LIN {X 0,Y 200.073,Z 515.512,A -85,B 0,C 180,E1 -21845.07,E2 -21845.07} C_VEL
LIN {X 0,Y 196.542,Z 522.437,A -85,B 0,C 180,E1 -21849.049,E2 -21849.049} C_VEL
LIN {X 0,Y 193.866,Z 527.871,A -85,B 0,C 180,E1 -21853.142,E2 -21853.142} C_VEL
LIN {X 0,Y 192.041,Z 531.966,A -85,B 0,C 180,E1 -21857.316,E2 -21857.316} C_VEL
LIN {X 0,Y 190.931,Z 534.837,A -85,B 0,C 180,E1 -21861.533,E2 -21861.533} C_VEL
LIN {X 0,Y 190.385,Z 536.558,A -85,B 0,C 180,E1 -21865.766,E2 -21865.766} C_VEL
LIN {X 0,Y 190.301,Z 537.156,A -85,B 0,C 180,E1 -21870,E2 -21870} C_VEL
LIN {X 0,Y 190.444,Z 536.444,A -85,B 0,C 180,E1 -21874.869,E2 -21874.869} C_VEL
LIN {X 0,Y 190.924,Z 534.92,A -85,B 0,C 180,E1 -21878.467,E2 -21878.467} C_VEL
LIN {X 0,Y 192.016,Z 532.092,A -85,B 0,C 180,E1 -21882.686,E2 -21882.686} C_VEL
LIN {X 0,Y 193.842,Z 528.039,A -85,B 0,C 180,E1 -21886.861,E2 -21886.861} C_VEL
LIN {X 0,Y 196.544,Z 522.658,A -85,B 0,C 180,E1 -21890.951,E2 -21890.951} C_VEL
LIN {X 0,Y 199.996,Z 515.797,A -85,B 0,C 180,E1 -21894.941,E2 -21894.941} C_VEL
LIN {X 0,Y 204.38,Z 507.224,A -85,B 0,C 180,E1 -21898.777,E2 -21898.777} C_VEL
LIN {X 0,Y 208.207,Z 499.512,A -85,B 0,C 180,E1 -21901.546,E2 -21901.546} C_VEL
LIN {X 0,Y 212.272,Z 490.435,A -85,B 0,C 180,E1 -21904.252,E2 -21904.252} C_VEL
LIN {X 0,Y 216.99,Z 479.715,A -85,B 0,C 180,E1 -21906.811,E2 -21906.811} C_VEL
LIN {X 0,Y 221.502,Z 468.012,A -85,B 0,C 180,E1 -21909.094,E2 -21909.094} C_VEL
LIN {X 0,Y 226.056,Z 455.219,A -85,B 0,C 180,E1 -21911.053,E2 -21911.053} C_VEL
LIN {X 0,Y 229.873,Z 442.172,A -85,B 0,C 180,E1 -21912.681,E2 -21912.681} C_VEL
LIN {X 0,Y 233.233,Z 428.457,A -85,B 0,C 180,E1 -21914.021,E2 -21914.021} C_VEL
LIN {X 0,Y 236.191,Z 413.431,A -85,B 0,C 180,E1 -21915.116,E2 -21915.116} C_VEL
LIN {X 0,Y 238.192,Z 399.868,A -85,B 0,C 180,E1 -21915.835,E2 -21915.835} C_VEL
LIN {X 0,Y 239.696,Z 384.094,A -85,B 0,C 180,E1 -21916.372,E2 -21916.372} C_VEL
LIN {X 0,Y 244.254,Z 312.757,A -85,B 0,C 180,E1 -21918.264,E2 -21918.264} C_VEL
LIN {X 0,Y 244.009,Z 311.507,A -85,B 0,C 180,E1 -21918.383,E2 -21918.383} C_VEL
LIN {X 0,Y 240.206,Z 303.509,A -85,B 0,C 180,E1 -21919.784,E2 -21919.784} C_VEL
LIN {X 0,Y 232.844,Z 290.889,A -85,B 0,C 180,E1 -21922.617,E2 -21922.617} C_VEL
LIN {X 0,Y 226.849,Z 281.57,A -85,B 0,C 180,E1 -21925.165,E2 -21925.165} C_VEL
LIN {X 0,Y 221.021,Z 273.151,A -85,B 0,C 180,E1 -21927.918,E2 -21927.918} C_VEL
LIN {X 0,Y 217.818,Z 268.869,A -85,B 0,C 180,E1 -21929.572,E2 -21929.572} C_VEL
LIN {X 0,Y 214.771,Z 264.799,A -85,B 0,C 180,E1 -21931.274,E2 -21931.274} C_VEL
LIN {X 0,Y 211.832,Z 260.873,A -85,B 0,C 180,E1 -21933.059,E2 -21933.059} C_VEL
LIN {X 0,Y 208.609,Z 257.265,A -85,B 0,C 180,E1 -21935.161,E2 -21935.161} C_VEL
LIN {X 0,Y 207.468,Z 255.378,A -85,B 0,C 180,E1 -21936.015,E2 -21936.015} C_VEL
LIN {X 0,Y 204.837,Z 253.006,A -85,B 0,C 180,E1 -21937.959,E2 -21937.959} C_VEL
LIN {X 0,Y 203.12,Z 250.05,A -85,B 0,C 180,E1 -21939.492,E2 -21939.492} C_VEL
LIN {X 0,Y 200.172,Z 247.881,A -85,B 0,C 180,E1 -21942.158,E2 -21942.158} C_VEL
LIN {X 0,Y 198.485,Z 244.934,A -85,B 0,C 180,E1 -21944.139,E2 -21944.139} C_VEL
LIN {X 0,Y 198.171,Z 244.119,A -85,B 0,C 180,E1 -21944.574,E2 -21944.574} C_VEL
LIN {X 0,Y 195.148,Z 242.441,A -85,B 0,C 180,E1 -21948.575,E2 -21948.575} C_VEL
LIN {X 0,Y 193.097,Z 238.68,A -85,B 0,C 180,E1 -21953.338,E2 -21953.338} C_VEL
LIN {X 0,Y 192.983,Z 238.059,A -85,B 0,C 180,E1 -21953.99,E2 -21953.99} C_VEL
LIN {X 0,Y 193.259,Z 238.03,A -85,B 0,C 180,E1 -21957.916,E2 -21957.916} C_VEL
LIN {X 0,Y 193.439,Z 238,A -85,B 0,C 180,E1 -21960,E2 -21960} C_VEL
LIN {X 0,Y 192.97,Z 238.063,A -85,B 0,C 180,E1 -21965.224,E2 -21965.224} C_VEL
LIN {X 0,Y 193.024,Z 238.361,A -85,B 0,C 180,E1 -21966.008,E2 -21966.008} C_VEL
LIN {X 0,Y 193.993,Z 240.918,A -85,B 0,C 180,E1 -21968.857,E2 -21968.857} C_VEL
LIN {X 0,Y 196.391,Z 243.419,A -85,B 0,C 180,E1 -21972.924,E2 -21972.924} C_VEL
LIN {X 0,Y 198.288,Z 244.285,A -85,B 0,C 180,E1 -21975.218,E2 -21975.218} C_VEL
LIN {X 0,Y 199.52,Z 246.969,A -85,B 0,C 180,E1 -21976.782,E2 -21976.782} C_VEL
LIN {X 0,Y 201.819,Z 249.303,A -85,B 0,C 180,E1 -21979.054,E2 -21979.054} C_VEL
LIN {X 0,Y 203.197,Z 250.271,A -85,B 0,C 180,E1 -21980.235,E2 -21980.235} C_VEL
LIN {X 0,Y 205.075,Z 253.32,A -85,B 0,C 180,E1 -21981.881,E2 -21981.881} C_VEL
LIN {X 0,Y 207.77,Z 255.795,A -85,B 0,C 180,E1 -21983.855,E2 -21983.855} C_VEL
LIN {X 0,Y 210.247,Z 259.306,A -85,B 0,C 180,E1 -21985.599,E2 -21985.599} C_VEL
LIN {X 0,Y 211.925,Z 261.053,A -85,B 0,C 180,E1 -21986.651,E2 -21986.651} C_VEL
LIN {X 0,Y 214.891,Z 264.939,A -85,B 0,C 180,E1 -21988.442,E2 -21988.442} C_VEL
LIN {X 0,Y 219.275,Z 270.946,A -85,B 0,C 180,E1 -21990.851,E2 -21990.851} C_VEL
LIN {X 0,Y 223.639,Z 278.116,A -85,B 0,C 180,E1 -21993.076,E2 -21993.076} C_VEL
LIN {X 0,Y 225.439,Z 282.403,A -85,B 0,C 180,E1 -21994.007,E2 -21994.007} C_VEL
LIN {X 0,Y 227.675,Z 290.656,A -85,B 0,C 180,E1 -21995.269,E2 -21995.269} C_VEL
LIN {X 0,Y 230.291,Z 300.869,A -85,B 0,C 180,E1 -21996.696,E2 -21996.696} C_VEL
LIN {X 0,Y 231.447,Z 304.009,A -85,B 0,C 180,E1 -21997.233,E2 -21997.233} C_VEL
LIN {X 0,Y 237.324,Z 317.3,A -85,B 0,C 180,E1 -21999.67,E2 -21999.67} C_VEL
LIN {X 0,Y 239.071,Z 321.76,A -85,B 0,C 180,E1 -22000.371,E2 -22000.371} C_VEL
LIN {X 0,Y 233.65,Z 401.493,A -85,B 0,C 180,E1 -22002.53,E2 -22002.53} C_VEL
LIN {X 0,Y 231.461,Z 417.617,A -85,B 0,C 180,E1 -22003.222,E2 -22003.222} C_VEL
LIN {X 0,Y 228.483,Z 432.859,A -85,B 0,C 180,E1 -22004.188,E2 -22004.188} C_VEL
LIN {X 0,Y 224.984,Z 446.59,A -85,B 0,C 180,E1 -22005.345,E2 -22005.345} C_VEL
LIN {X 0,Y 220.786,Z 460.673,A -85,B 0,C 180,E1 -22006.939,E2 -22006.939} C_VEL
LIN {X 0,Y 215.719,Z 474.962,A -85,B 0,C 180,E1 -22009.031,E2 -22009.031} C_VEL
LIN {X 0,Y 210.669,Z 487.181,A -85,B 0,C 180,E1 -22011.282,E2 -22011.282} C_VEL
LIN {X 0,Y 205.703,Z 498.349,A -85,B 0,C 180,E1 -22013.89,E2 -22013.89} C_VEL
LIN {X 0,Y 201.078,Z 507.901,A -85,B 0,C 180,E1 -22016.66,E2 -22016.66} C_VEL
LIN {X 0,Y 196.607,Z 517.011,A -85,B 0,C 180,E1 -22019.971,E2 -22019.971} C_VEL
LIN {X 0,Y 192.032,Z 525.729,A -85,B 0,C 180,E1 -22023.949,E2 -22023.949} C_VEL
LIN {X 0,Y 188.457,Z 532.733,A -85,B 0,C 180,E1 -22028.105,E2 -22028.105} C_VEL
LIN {X 0,Y 185.854,Z 538.249,A -85,B 0,C 180,E1 -22032.392,E2 -22032.392} C_VEL
LIN {X 0,Y 184.088,Z 542.425,A -85,B 0,C 180,E1 -22036.758,E2 -22036.758} C_VEL
LIN {X 0,Y 183.224,Z 545.362,A -85,B 0,C 180,E1 -22041.174,E2 -22041.174} C_VEL
LIN {X 0,Y 182.976,Z 547.117,A -85,B 0,C 180,E1 -22045.594,E2 -22045.594} C_VEL
LIN {X 0,Y 183.168,Z 547.723,A -85,B 0,C 180,E1 -22050,E2 -22050} C_VEL
LIN {X 0,Y 182.976,Z 547.101,A -85,B 0,C 180,E1 -22054.406,E2 -22054.406} C_VEL
LIN {X 0,Y 183.224,Z 545.325,A -85,B 0,C 180,E1 -22058.826,E2 -22058.826} C_VEL
LIN {X 0,Y 184.079,Z 542.372,A -85,B 0,C 180,E1 -22063.242,E2 -22063.242} C_VEL
LIN {X 0,Y 185.809,Z 538.181,A -85,B 0,C 180,E1 -22067.613,E2 -22067.613} C_VEL
LIN {X 0,Y 188.416,Z 532.64,A -85,B 0,C 180,E1 -22071.9,E2 -22071.9} C_VEL
LIN {X 0,Y 192.024,Z 525.605,A -85,B 0,C 180,E1 -22076.052,E2 -22076.052} C_VEL
LIN {X 0,Y 196.602,Z 516.864,A -85,B 0,C 180,E1 -22080.03,E2 -22080.03} C_VEL
LIN {X 0,Y 200.433,Z 509.032,A -85,B 0,C 180,E1 -22082.92,E2 -22082.92} C_VEL
LIN {X 0,Y 205.673,Z 498.149,A -85,B 0,C 180,E1 -22086.117,E2 -22086.117} C_VEL
LIN {X 0,Y 211.098,Z 485.92,A -85,B 0,C 180,E1 -22088.931,E2 -22088.931} C_VEL
LIN {X 0,Y 216.164,Z 473.554,A -85,B 0,C 180,E1 -22091.152,E2 -22091.152} C_VEL
LIN {X 0,Y 220.965,Z 459.667,A -85,B 0,C 180,E1 -22093.141,E2 -22093.141} C_VEL
LIN {X 0,Y 225.004,Z 446.104,A -85,B 0,C 180,E1 -22094.65,E2 -22094.65} C_VEL
LIN {X 0,Y 228.45,Z 432.306,A -85,B 0,C 180,E1 -22095.821,E2 -22095.821} C_VEL
LIN {X 0,Y 231.449,Z 416.84,A -85,B 0,C 180,E1 -22096.781,E2 -22096.781} C_VEL
LIN {X 0,Y 233.503,Z 401.515,A -85,B 0,C 180,E1 -22097.429,E2 -22097.429} C_VEL
LIN {X 0,Y 238.923,Z 321.559,A -85,B 0,C 180,E1 -22099.598,E2 -22099.598} C_VEL
LIN {X 0,Y 233.667,Z 309.004,A -85,B 0,C 180,E1 -22101.728,E2 -22101.728} C_VEL
LIN {X 0,Y 228.26,Z 297.683,A -85,B 0,C 180,E1 -22104.056,E2 -22104.056} C_VEL
LIN {X 0,Y 221.561,Z 285.075,A -85,B 0,C 180,E1 -22107.226,E2 -22107.226} C_VEL
LIN {X 0,Y 215.675,Z 275.329,A -85,B 0,C 180,E1 -22110.35,E2 -22110.35} C_VEL
LIN {X 0,Y 212.532,Z 271.116,A -85,B 0,C 180,E1 -22112.155,E2 -22112.155} C_VEL
LIN {X 0,Y 209.049,Z 266.549,A -85,B 0,C 180,E1 -22114.352,E2 -22114.352} C_VEL
LIN {X 0,Y 206.238,Z 263.031,A -85,B 0,C 180,E1 -22116.306,E2 -22116.306} C_VEL
LIN {X 0,Y 205.38,Z 261.817,A -85,B 0,C 180,E1 -22116.957,E2 -22116.957} C_VEL
LIN {X 0,Y 202.667,Z 259.01,A -85,B 0,C 180,E1 -22119.08,E2 -22119.08} C_VEL
LIN {X 0,Y 201.289,Z 256.619,A -85,B 0,C 180,E1 -22120.363,E2 -22120.363} C_VEL
LIN {X 0,Y 198.829,Z 254.709,A -85,B 0,C 180,E1 -22122.652,E2 -22122.652} C_VEL
LIN {X 0,Y 197.011,Z 251.645,A -85,B 0,C 180,E1 -22124.813,E2 -22124.813} C_VEL
LIN {X 0,Y 196.685,Z 251.002,A -85,B 0,C 180,E1 -22125.251,E2 -22125.251} C_VEL
LIN {X 0,Y 193.835,Z 249.178,A -85,B 0,C 180,E1 -22129.159,E2 -22129.159} C_VEL
LIN {X 0,Y 192.101,Z 245.791,A -85,B 0,C 180,E1 -22133.172,E2 -22133.172} C_VEL
LIN {X 0,Y 191.964,Z 245.215,A -85,B 0,C 180,E1 -22133.695,E2 -22133.695} C_VEL
LIN {X 0,Y 190.797,Z 244.592,A -85,B 0,C 180,E1 -22140,E2 -22140} C_VEL
LIN {X 0,Y 192.02,Z 245.3,A -85,B 0,C 180,E1 -22146.922,E2 -22146.922} C_VEL
LIN {X 0,Y 193.208,Z 248.355,A -85,B 0,C 180,E1 -22150.116,E2 -22150.116} C_VEL
LIN {X 0,Y 195.519,Z 250.483,A -85,B 0,C 180,E1 -22153.777,E2 -22153.777} C_VEL
LIN {X 0,Y 196.859,Z 251.175,A -85,B 0,C 180,E1 -22155.404,E2 -22155.404} C_VEL
LIN {X 0,Y 198.617,Z 254.503,A -85,B 0,C 180,E1 -22157.573,E2 -22157.573} C_VEL
LIN {X 0,Y 201.561,Z 257.081,A -85,B 0,C 180,E1 -22160.34,E2 -22160.34} C_VEL
LIN {X 0,Y 203.639,Z 260.282,A -85,B 0,C 180,E1 -22162.178,E2 -22162.178} C_VEL
LIN {X 0,Y 205.868,Z 262.39,A -85,B 0,C 180,E1 -22163.849,E2 -22163.849} C_VEL
LIN {X 0,Y 208.483,Z 265.974,A -85,B 0,C 180,E1 -22165.723,E2 -22165.723} C_VEL
LIN {X 0,Y 209.926,Z 267.715,A -85,B 0,C 180,E1 -22166.668,E2 -22166.668} C_VEL
LIN {X 0,Y 213.752,Z 272.8,A -85,B 0,C 180,E1 -22169.011,E2 -22169.011} C_VEL
LIN {X 0,Y 217.656,Z 278.21,A -85,B 0,C 180,E1 -22171.17,E2 -22171.17} C_VEL
LIN {X 0,Y 222.126,Z 284.657,A -85,B 0,C 180,E1 -22173.417,E2 -22173.417} C_VEL
LIN {X 0,Y 228.603,Z 294.778,A -85,B 0,C 180,E1 -22176.354,E2 -22176.354} C_VEL
LIN {X 0,Y 235.567,Z 306.886,A -85,B 0,C 180,E1 -22179.192,E2 -22179.192} C_VEL
LIN {X 0,Y 238.998,Z 313.895,A -85,B 0,C 180,E1 -22180.518,E2 -22180.518} C_VEL
LIN {X 0,Y 239.319,Z 314.642,A -85,B 0,C 180,E1 -22180.642,E2 -22180.642} C_VEL
LIN {X 0,Y 234.099,Z 391.732,A -85,B 0,C 180,E1 -22182.729,E2 -22182.729} C_VEL
LIN {X 0,Y 232.159,Z 407.333,A -85,B 0,C 180,E1 -22183.405,E2 -22183.405} C_VEL
LIN {X 0,Y 229.304,Z 422.917,A -85,B 0,C 180,E1 -22184.398,E2 -22184.398} C_VEL
LIN {X 0,Y 225.844,Z 437.614,A -85,B 0,C 180,E1 -22185.704,E2 -22185.704} C_VEL
LIN {X 0,Y 221.823,Z 451.806,A -85,B 0,C 180,E1 -22187.374,E2 -22187.374} C_VEL
LIN {X 0,Y 217.107,Z 465.249,A -85,B 0,C 180,E1 -22189.349,E2 -22189.349} C_VEL
LIN {X 0,Y 212.275,Z 477.449,A -85,B 0,C 180,E1 -22191.628,E2 -22191.628} C_VEL
LIN {X 0,Y 207.309,Z 488.564,A -85,B 0,C 180,E1 -22194.213,E2 -22194.213} C_VEL
LIN {X 0,Y 202.282,Z 499.345,A -85,B 0,C 180,E1 -22197.417,E2 -22197.417} C_VEL
LIN {X 0,Y 197.612,Z 508.3,A -85,B 0,C 180,E1 -22200.725,E2 -22200.725} C_VEL
LIN {X 0,Y 193.632,Z 515.715,A -85,B 0,C 180,E1 -22204.181,E2 -22204.181} C_VEL
LIN {X 0,Y 189.896,Z 522.64,A -85,B 0,C 180,E1 -22208.279,E2 -22208.279} C_VEL
LIN {X 0,Y 187.065,Z 528.074,A -85,B 0,C 180,E1 -22212.509,E2 -22212.509} C_VEL
LIN {X 0,Y 185.108,Z 532.168,A -85,B 0,C 180,E1 -22216.833,E2 -22216.833} C_VEL
LIN {X 0,Y 183.885,Z 535.039,A -85,B 0,C 180,E1 -22221.206,E2 -22221.206} C_VEL
LIN {X 0,Y 183.308,Z 536.759,A -85,B 0,C 180,E1 -22225.602,E2 -22225.602} C_VEL
LIN {X 0,Y 183.207,Z 537.356,A -85,B 0,C 180,E1 -22230,E2 -22230} C_VEL
LIN {X 0,Y 183.331,Z 536.742,A -85,B 0,C 180,E1 -22234.644,E2 -22234.644} C_VEL
LIN {X 0,Y 183.876,Z 535.121,A -85,B 0,C 180,E1 -22238.794,E2 -22238.794} C_VEL
LIN {X 0,Y 185.082,Z 532.293,A -85,B 0,C 180,E1 -22243.169,E2 -22243.169} C_VEL
LIN {X 0,Y 187.042,Z 528.24,A -85,B 0,C 180,E1 -22247.493,E2 -22247.493} C_VEL
LIN {X 0,Y 189.905,Z 522.858,A -85,B 0,C 180,E1 -22251.72,E2 -22251.72} C_VEL
LIN {X 0,Y 193.546,Z 515.997,A -85,B 0,C 180,E1 -22255.832,E2 -22255.832} C_VEL
LIN {X 0,Y 198.15,Z 507.424,A -85,B 0,C 180,E1 -22259.771,E2 -22259.771} C_VEL
LIN {X 0,Y 202.87,Z 498.302,A -85,B 0,C 180,E1 -22263.067,E2 -22263.067} C_VEL
LIN {X 0,Y 207.223,Z 489.015,A -85,B 0,C 180,E1 -22265.805,E2 -22265.805} C_VEL
LIN {X 0,Y 212.634,Z 476.978,A -85,B 0,C 180,E1 -22268.597,E2 -22268.597} C_VEL
LIN {X 0,Y 216.98,Z 465.87,A -85,B 0,C 180,E1 -22270.68,E2 -22270.68} C_VEL
LIN {X 0,Y 221.68,Z 452.576,A -85,B 0,C 180,E1 -22272.66,E2 -22272.66} C_VEL
LIN {X 0,Y 225.562,Z 439.157,A -85,B 0,C 180,E1 -22274.265,E2 -22274.265} C_VEL
LIN {X 0,Y 228.955,Z 425.268,A -85,B 0,C 180,E1 -22275.534,E2 -22275.534} C_VEL
LIN {X 0,Y 231.728,Z 410.581,A -85,B 0,C 180,E1 -22276.55,E2 -22276.55} C_VEL
LIN {X 0,Y 233.869,Z 395.505,A -85,B 0,C 180,E1 -22277.253,E2 -22277.253} C_VEL
LIN {X 0,Y 235.609,Z 373.547,A -85,B 0,C 180,E1 -22277.9,E2 -22277.9} C_VEL
LIN {X 0,Y 239.465,Z 314.745,A -85,B 0,C 180,E1 -22279.483,E2 -22279.483} C_VEL
LIN {X 0,Y 236.074,Z 307.675,A -85,B 0,C 180,E1 -22280.795,E2 -22280.795} C_VEL
LIN {X 0,Y 229.277,Z 295.796,A -85,B 0,C 180,E1 -22283.553,E2 -22283.553} C_VEL
LIN {X 0,Y 223.708,Z 286.964,A -85,B 0,C 180,E1 -22286.04,E2 -22286.04} C_VEL
LIN {X 0,Y 218.195,Z 278.792,A -85,B 0,C 180,E1 -22288.776,E2 -22288.776} C_VEL
LIN {X 0,Y 214.914,Z 274.378,A -85,B 0,C 180,E1 -22290.556,E2 -22290.556} C_VEL
LIN {X 0,Y 212.264,Z 270.742,A -85,B 0,C 180,E1 -22292.116,E2 -22292.116} C_VEL
LIN {X 0,Y 208.991,Z 266.469,A -85,B 0,C 180,E1 -22294.207,E2 -22294.207} C_VEL
LIN {X 0,Y 206.184,Z 262.882,A -85,B 0,C 180,E1 -22296.19,E2 -22296.19} C_VEL
LIN {X 0,Y 205.35,Z 261.788,A -85,B 0,C 180,E1 -22296.822,E2 -22296.822} C_VEL
LIN {X 0,Y 202.512,Z 258.694,A -85,B 0,C 180,E1 -22299.096,E2 -22299.096} C_VEL
LIN {X 0,Y 201.24,Z 256.617,A -85,B 0,C 180,E1 -22300.292,E2 -22300.292} C_VEL
LIN {X 0,Y 198.616,Z 254.402,A -85,B 0,C 180,E1 -22302.817,E2 -22302.817} C_VEL
LIN {X 0,Y 196.92,Z 251.309,A -85,B 0,C 180,E1 -22304.938,E2 -22304.938} C_VEL
LIN {X 0,Y 193.608,Z 248.789,A -85,B 0,C 180,E1 -22309.745,E2 -22309.745} C_VEL
LIN {X 0,Y 191.993,Z 245.077,A -85,B 0,C 180,E1 -22314.222,E2 -22314.222} C_VEL
LIN {X 0,Y 191.256,Z 244.85,A -85,B 0,C 180,E1 -22322.106,E2 -22322.106} C_VEL
LIN {X 0,Y 192,Z 245.258,A -85,B 0,C 180,E1 -22325.514,E2 -22325.514} C_VEL
LIN {X 0,Y 193.763,Z 249.03,A -85,B 0,C 180,E1 -22330.206,E2 -22330.206} C_VEL
LIN {X 0,Y 196.329,Z 250.872,A -85,B 0,C 180,E1 -22333.983,E2 -22333.983} C_VEL
LIN {X 0,Y 196.934,Z 251.343,A -85,B 0,C 180,E1 -22334.73,E2 -22334.73} C_VEL
LIN {X 0,Y 198.513,Z 254.249,A -85,B 0,C 180,E1 -22336.713,E2 -22336.713} C_VEL
LIN {X 0,Y 200.988,Z 256.462,A -85,B 0,C 180,E1 -22339.136,E2 -22339.136} C_VEL
LIN {X 0,Y 201.614,Z 257.144,A -85,B 0,C 180,E1 -22339.707,E2 -22339.707} C_VEL
LIN {X 0,Y 203.926,Z 260.514,A -85,B 0,C 180,E1 -22341.745,E2 -22341.745} C_VEL
LIN {X 0,Y 205.907,Z 262.38,A -85,B 0,C 180,E1 -22343.238,E2 -22343.238} C_VEL
LIN {X 0,Y 208.586,Z 266.064,A -85,B 0,C 180,E1 -22345.175,E2 -22345.175} C_VEL
LIN {X 0,Y 210.023,Z 267.779,A -85,B 0,C 180,E1 -22346.119,E2 -22346.119} C_VEL
LIN {X 0,Y 214.104,Z 273.215,A -85,B 0,C 180,E1 -22348.623,E2 -22348.623} C_VEL
LIN {X 0,Y 216.638,Z 276.831,A -85,B 0,C 180,E1 -22350.053,E2 -22350.053} C_VEL
LIN {X 0,Y 222.332,Z 286.445,A -85,B 0,C 180,E1 -22353.043,E2 -22353.043} C_VEL
LIN {X 0,Y 228.743,Z 298.538,A -85,B 0,C 180,E1 -22356.055,E2 -22356.055} C_VEL
LIN {X 0,Y 231.447,Z 304.009,A -85,B 0,C 180,E1 -22357.233,E2 -22357.233} C_VEL
LIN {X 0,Y 232.971,Z 308.912,A -85,B 0,C 180,E1 -22357.961,E2 -22357.961} C_VEL
LIN {X 0,Y 234.004,Z 316.28,A -85,B 0,C 180,E1 -22358.637,E2 -22358.637} C_VEL
LIN {X 0,Y 234.134,Z 326.178,A -85,B 0,C 180,E1 -22359.148,E2 -22359.148} C_VEL
LIN {X 0,Y 233.722,Z 334.247,A -85,B 0,C 180,E1 -22359.407,E2 -22359.407} C_VEL
LIN {X 0,Y 228.917,Z 401.309,A -85,B 0,C 180,E1 -22361.222,E2 -22361.222} C_VEL
LIN {X 0,Y 226.649,Z 417.425,A -85,B 0,C 180,E1 -22361.911,E2 -22361.911} C_VEL
LIN {X 0,Y 223.595,Z 432.665,A -85,B 0,C 180,E1 -22362.884,E2 -22362.884} C_VEL
LIN {X 0,Y 219.991,Z 446.395,A -85,B 0,C 180,E1 -22364.046,E2 -22364.046} C_VEL
LIN {X 0,Y 215.82,Z 459.857,A -85,B 0,C 180,E1 -22365.565,E2 -22365.565} C_VEL
LIN {X 0,Y 210.827,Z 473.757,A -85,B 0,C 180,E1 -22367.594,E2 -22367.594} C_VEL
LIN {X 0,Y 205.585,Z 485.971,A -85,B 0,C 180,E1 -22369.817,E2 -22369.817} C_VEL
LIN {X 0,Y 199.957,Z 498.149,A -85,B 0,C 180,E1 -22372.679,E2 -22372.679} C_VEL
LIN {X 0,Y 194.456,Z 508.987,A -85,B 0,C 180,E1 -22375.931,E2 -22375.931} C_VEL
LIN {X 0,Y 189.8,Z 518.027,A -85,B 0,C 180,E1 -22379.394,E2 -22379.394} C_VEL
LIN {X 0,Y 185.592,Z 525.527,A -85,B 0,C 180,E1 -22382.973,E2 -22382.973} C_VEL
LIN {X 0,Y 181.808,Z 532.531,A -85,B 0,C 180,E1 -22387.26,E2 -22387.26} C_VEL
LIN {X 0,Y 179.04,Z 538.048,A -85,B 0,C 180,E1 -22391.698,E2 -22391.698} C_VEL
LIN {X 0,Y 177.123,Z 542.223,A -85,B 0,C 180,E1 -22396.228,E2 -22396.228} C_VEL
LIN {X 0,Y 176.18,Z 545.16,A -85,B 0,C 180,E1 -22400.819,E2 -22400.819} C_VEL
LIN {X 0,Y 175.876,Z 546.916,A -85,B 0,C 180,E1 -22405.416,E2 -22405.416} C_VEL
LIN {X 0,Y 176.074,Z 547.522,A -85,B 0,C 180,E1 -22410,E2 -22410} C_VEL
LIN {X 0,Y 175.876,Z 546.9,A -85,B 0,C 180,E1 -22414.584,E2 -22414.584} C_VEL
LIN {X 0,Y 176.18,Z 545.123,A -85,B 0,C 180,E1 -22419.181,E2 -22419.181} C_VEL
LIN {X 0,Y 177.111,Z 542.169,A -85,B 0,C 180,E1 -22423.773,E2 -22423.773} C_VEL
LIN {X 0,Y 178.991,Z 537.977,A -85,B 0,C 180,E1 -22428.307,E2 -22428.307} C_VEL
LIN {X 0,Y 181.772,Z 532.436,A -85,B 0,C 180,E1 -22432.745,E2 -22432.745} C_VEL
LIN {X 0,Y 185.586,Z 525.4,A -85,B 0,C 180,E1 -22437.028,E2 -22437.028} C_VEL
LIN {X 0,Y 189.795,Z 517.886,A -85,B 0,C 180,E1 -22440.607,E2 -22440.607} C_VEL
LIN {X 0,Y 194.462,Z 508.824,A -85,B 0,C 180,E1 -22444.068,E2 -22444.068} C_VEL
LIN {X 0,Y 199.924,Z 497.943,A -85,B 0,C 180,E1 -22447.328,E2 -22447.328} C_VEL
LIN {X 0,Y 205.569,Z 485.714,A -85,B 0,C 180,E1 -22450.187,E2 -22450.187} C_VEL
LIN {X 0,Y 210.778,Z 473.55,A -85,B 0,C 180,E1 -22452.393,E2 -22452.393} C_VEL
LIN {X 0,Y 215.245,Z 461.14,A -85,B 0,C 180,E1 -22454.225,E2 -22454.225} C_VEL
LIN {X 0,Y 219.467,Z 447.739,A -85,B 0,C 180,E1 -22455.766,E2 -22455.766} C_VEL
LIN {X 0,Y 223.256,Z 433.235,A -85,B 0,C 180,E1 -22457.044,E2 -22457.044} C_VEL
LIN {X 0,Y 226.366,Z 418.199,A -85,B 0,C 180,E1 -22458.002,E2 -22458.002} C_VEL
LIN {X 0,Y 228.631,Z 402.487,A -85,B 0,C 180,E1 -22458.693,E2 -22458.693} C_VEL
LIN {X 0,Y 231.914,Z 357.932,A -85,B 0,C 180,E1 -22459.924,E2 -22459.924} C_VEL
LIN {X 0,Y 234.19,Z 323.957,A -85,B 0,C 180,E1 -22460.854,E2 -22460.854} C_VEL
LIN {X 0,Y 228.686,Z 310.84,A -85,B 0,C 180,E1 -22463.232,E2 -22463.232} C_VEL
LIN {X 0,Y 222.73,Z 298.519,A -85,B 0,C 180,E1 -22466.003,E2 -22466.003} C_VEL
LIN {X 0,Y 217.43,Z 288.611,A -85,B 0,C 180,E1 -22468.722,E2 -22468.722} C_VEL
LIN {X 0,Y 213.021,Z 281.156,A -85,B 0,C 180,E1 -22471.218,E2 -22471.218} C_VEL
LIN {X 0,Y 209.884,Z 276.878,A -85,B 0,C 180,E1 -22473.116,E2 -22473.116} C_VEL
LIN {X 0,Y 206.891,Z 272.784,A -85,B 0,C 180,E1 -22475.109,E2 -22475.109} C_VEL
LIN {X 0,Y 204.048,Z 268.987,A -85,B 0,C 180,E1 -22477.202,E2 -22477.202} C_VEL
LIN {X 0,Y 200.557,Z 264.897,A -85,B 0,C 180,E1 -22480.089,E2 -22480.089} C_VEL
LIN {X 0,Y 199.632,Z 263.306,A -85,B 0,C 180,E1 -22480.996,E2 -22480.996} C_VEL
LIN {X 0,Y 197.061,Z 260.984,A -85,B 0,C 180,E1 -22483.556,E2 -22483.556} C_VEL
LIN {X 0,Y 195.418,Z 257.897,A -85,B 0,C 180,E1 -22485.685,E2 -22485.685} C_VEL
LIN {X 0,Y 192.75,Z 256.101,A -85,B 0,C 180,E1 -22489.496,E2 -22489.496} C_VEL
LIN {X 0,Y 191.026,Z 252.491,A -85,B 0,C 180,E1 -22493.796,E2 -22493.796} C_VEL
LIN {X 0,Y 190.755,Z 252.094,A -85,B 0,C 180,E1 -22494.715,E2 -22494.715} C_VEL
LIN {X 0,Y 189.932,Z 251.639,A -85,B 0,C 180,E1 -22500,E2 -22500} C_VEL
LIN {X 0,Y 191.008,Z 252.227,A -85,B 0,C 180,E1 -22506.51,E2 -22506.51} C_VEL
LIN {X 0,Y 192.165,Z 255.317,A -85,B 0,C 180,E1 -22509.812,E2 -22509.812} C_VEL
LIN {X 0,Y 194.673,Z 257.583,A -85,B 0,C 180,E1 -22513.838,E2 -22513.838} C_VEL
LIN {X 0,Y 195.563,Z 258.237,A -85,B 0,C 180,E1 -22514.969,E2 -22514.969} C_VEL
LIN {X 0,Y 197.466,Z 261.535,A -85,B 0,C 180,E1 -22517.342,E2 -22517.342} C_VEL
LIN {X 0,Y 199.957,Z 263.83,A -85,B 0,C 180,E1 -22519.768,E2 -22519.768} C_VEL
LIN {X 0,Y 202.351,Z 267.299,A -85,B 0,C 180,E1 -22521.924,E2 -22521.924} C_VEL
LIN {X 0,Y 204.076,Z 269.043,A -85,B 0,C 180,E1 -22523.264,E2 -22523.264} C_VEL
LIN {X 0,Y 206.637,Z 272.505,A -85,B 0,C 180,E1 -22525.161,E2 -22525.161} C_VEL
LIN {X 0,Y 207.87,Z 274.097,A -85,B 0,C 180,E1 -22526.006,E2 -22526.006} C_VEL
LIN {X 0,Y 211.655,Z 279.318,A -85,B 0,C 180,E1 -22528.422,E2 -22528.422} C_VEL
LIN {X 0,Y 215.326,Z 284.46,A -85,B 0,C 180,E1 -22530.527,E2 -22530.527} C_VEL
LIN {X 0,Y 220.608,Z 292.431,A -85,B 0,C 180,E1 -22533.267,E2 -22533.267} C_VEL
LIN {X 0,Y 226.578,Z 302.199,A -85,B 0,C 180,E1 -22536.042,E2 -22536.042} C_VEL
LIN {X 0,Y 232.932,Z 313.73,A -85,B 0,C 180,E1 -22538.717,E2 -22538.717} C_VEL
LIN {X 0,Y 234.59,Z 317.241,A -85,B 0,C 180,E1 -22539.39,E2 -22539.39} C_VEL
LIN {X 0,Y 229.343,Z 391.993,A -85,B 0,C 180,E1 -22541.429,E2 -22541.429} C_VEL
LIN {X 0,Y 227.347,Z 407.545,A -85,B 0,C 180,E1 -22542.107,E2 -22542.107} C_VEL
LIN {X 0,Y 224.394,Z 423.126,A -85,B 0,C 180,E1 -22543.103,E2 -22543.103} C_VEL
LIN {X 0,Y 220.898,Z 437.539,A -85,B 0,C 180,E1 -22544.39,E2 -22544.39} C_VEL
LIN {X 0,Y 216.656,Z 452.011,A -85,B 0,C 180,E1 -22546.104,E2 -22546.104} C_VEL
LIN {X 0,Y 211.774,Z 465.454,A -85,B 0,C 180,E1 -22548.098,E2 -22548.098} C_VEL
LIN {X 0,Y 206.76,Z 477.652,A -85,B 0,C 180,E1 -22550.408,E2 -22550.408} C_VEL
LIN {X 0,Y 201.574,Z 488.768,A -85,B 0,C 180,E1 -22553.029,E2 -22553.029} C_VEL
LIN {X 0,Y 197.751,Z 496.629,A -85,B 0,C 180,E1 -22555.346,E2 -22555.346} C_VEL
LIN {X 0,Y 192.729,Z 506.068,A -85,B 0,C 180,E1 -22558.693,E2 -22558.693} C_VEL
LIN {X 0,Y 187.805,Z 514.919,A -85,B 0,C 180,E1 -22562.716,E2 -22562.716} C_VEL
LIN {X 0,Y 184.223,Z 521.116,A -85,B 0,C 180,E1 -22566.29,E2 -22566.29} C_VEL
LIN {X 0,Y 181.012,Z 527.047,A -85,B 0,C 180,E1 -22570.73,E2 -22570.73} C_VEL
LIN {X 0,Y 179.083,Z 530.484,A -85,B 0,C 180,E1 -22574.056,E2 -22574.056} C_VEL
LIN {X 0,Y 177.422,Z 533.953,A -85,B 0,C 180,E1 -22578.577,E2 -22578.577} C_VEL
LIN {X 0,Y 176.467,Z 536.241,A -85,B 0,C 180,E1 -22583.138,E2 -22583.138} C_VEL
LIN {X 0,Y 176.106,Z 537.403,A -85,B 0,C 180,E1 -22587.713,E2 -22587.713} C_VEL
LIN {X 0,Y 176.116,Z 537.557,A -85,B 0,C 180,E1 -22590,E2 -22590} C_VEL
LIN {X 0,Y 176.226,Z 536.995,A -85,B 0,C 180,E1 -22594.575,E2 -22594.575} C_VEL
LIN {X 0,Y 176.845,Z 535.322,A -85,B 0,C 180,E1 -22599.147,E2 -22599.147} C_VEL
LIN {X 0,Y 178.13,Z 532.494,A -85,B 0,C 180,E1 -22603.693,E2 -22603.693} C_VEL
LIN {X 0,Y 180.272,Z 528.44,A -85,B 0,C 180,E1 -22608.172,E2 -22608.172} C_VEL
LIN {X 0,Y 183.308,Z 523.058,A -85,B 0,C 180,E1 -22612.544,E2 -22612.544} C_VEL
LIN {X 0,Y 187.169,Z 516.197,A -85,B 0,C 180,E1 -22616.781,E2 -22616.781} C_VEL
LIN {X 0,Y 191.994,Z 507.623,A -85,B 0,C 180,E1 -22620.828,E2 -22620.828} C_VEL
LIN {X 0,Y 196.918,Z 498.502,A -85,B 0,C 180,E1 -22624.201,E2 -22624.201} C_VEL
LIN {X 0,Y 200.675,Z 490.832,A -85,B 0,C 180,E1 -22626.538,E2 -22626.538} C_VEL
LIN {X 0,Y 205.777,Z 480.111,A -85,B 0,C 180,E1 -22629.185,E2 -22629.185} C_VEL
LIN {X 0,Y 210.692,Z 468.405,A -85,B 0,C 180,E1 -22631.525,E2 -22631.525} C_VEL
LIN {X 0,Y 215.544,Z 455.612,A -85,B 0,C 180,E1 -22633.534,E2 -22633.534} C_VEL
LIN {X 0,Y 219.469,Z 443.109,A -85,B 0,C 180,E1 -22635.138,E2 -22635.138} C_VEL
LIN {X 0,Y 223.254,Z 428.843,A -85,B 0,C 180,E1 -22636.551,E2 -22636.551} C_VEL
LIN {X 0,Y 226.279,Z 414.573,A -85,B 0,C 180,E1 -22637.613,E2 -22637.613} C_VEL
LIN {X 0,Y 228.548,Z 400.241,A -85,B 0,C 180,E1 -22638.384,E2 -22638.384} C_VEL
LIN {X 0,Y 230.147,Z 384.448,A -85,B 0,C 180,E1 -22638.926,E2 -22638.926} C_VEL
LIN {X 0,Y 234.801,Z 317.457,A -85,B 0,C 180,E1 -22640.713,E2 -22640.713} C_VEL
LIN {X 0,Y 230.576,Z 309.145,A -85,B 0,C 180,E1 -22642.439,E2 -22642.439} C_VEL
LIN {X 0,Y 223.454,Z 296.728,A -85,B 0,C 180,E1 -22645.587,E2 -22645.587} C_VEL
LIN {X 0,Y 216.316,Z 285.665,A -85,B 0,C 180,E1 -22649.172,E2 -22649.172} C_VEL
LIN {X 0,Y 210.426,Z 277.402,A -85,B 0,C 180,E1 -22652.595,E2 -22652.595} C_VEL
LIN {X 0,Y 207.04,Z 272.939,A -85,B 0,C 180,E1 -22654.832,E2 -22654.832} C_VEL
LIN {X 0,Y 204.108,Z 269.007,A -85,B 0,C 180,E1 -22657.008,E2 -22657.008} C_VEL
LIN {X 0,Y 200.649,Z 264.948,A -85,B 0,C 180,E1 -22659.898,E2 -22659.898} C_VEL
LIN {X 0,Y 199.8,Z 263.412,A -85,B 0,C 180,E1 -22660.745,E2 -22660.745} C_VEL
LIN {X 0,Y 197.239,Z 261.191,A -85,B 0,C 180,E1 -22663.304,E2 -22663.304} C_VEL
LIN {X 0,Y 195.424,Z 257.881,A -85,B 0,C 180,E1 -22665.685,E2 -22665.685} C_VEL
LIN {X 0,Y 192.841,Z 256.126,A -85,B 0,C 180,E1 -22669.501,E2 -22669.501} C_VEL
LIN {X 0,Y 190.969,Z 252.109,A -85,B 0,C 180,E1 -22674.721,E2 -22674.721} C_VEL
LIN {X 0,Y 190.393,Z 251.877,A -85,B 0,C 180,E1 -22682.115,E2 -22682.115} C_VEL
LIN {X 0,Y 191.02,Z 252.238,A -85,B 0,C 180,E1 -22685.145,E2 -22685.145} C_VEL
LIN {X 0,Y 192.773,Z 256.038,A -85,B 0,C 180,E1 -22690.016,E2 -22690.016} C_VEL
LIN {X 0,Y 195.572,Z 258.136,A -85,B 0,C 180,E1 -22694.17,E2 -22694.17} C_VEL
LIN {X 0,Y 197.206,Z 261.095,A -85,B 0,C 180,E1 -22696.299,E2 -22696.299} C_VEL
LIN {X 0,Y 200.056,Z 263.876,A -85,B 0,C 180,E1 -22699.162,E2 -22699.162} C_VEL
LIN {X 0,Y 202.349,Z 267.214,A -85,B 0,C 180,E1 -22701.255,E2 -22701.255} C_VEL
LIN {X 0,Y 204.255,Z 269.249,A -85,B 0,C 180,E1 -22702.758,E2 -22702.758} C_VEL
LIN {X 0,Y 207.221,Z 273.091,A -85,B 0,C 180,E1 -22704.934,E2 -22704.934} C_VEL
LIN {X 0,Y 211.765,Z 279.361,A -85,B 0,C 180,E1 -22707.887,E2 -22707.887} C_VEL
LIN {X 0,Y 214.244,Z 283.071,A -85,B 0,C 180,E1 -22709.355,E2 -22709.355} C_VEL
LIN {X 0,Y 219.28,Z 291.818,A -85,B 0,C 180,E1 -22712.129,E2 -22712.129} C_VEL
LIN {X 0,Y 225.221,Z 303.293,A -85,B 0,C 180,E1 -22715.072,E2 -22715.072} C_VEL
LIN {X 0,Y 230.347,Z 314.401,A -85,B 0,C 180,E1 -22717.398,E2 -22717.398} C_VEL
LIN {X 0,Y 234.338,Z 324.148,A -85,B 0,C 180,E1 -22719.113,E2 -22719.113} C_VEL
LIN {X 0,Y 233.722,Z 334.247,A -85,B 0,C 180,E1 -22719.407,E2 -22719.407} C_VEL
LIN {X 0,Y 232.902,Z 340.098,A -85,B 0,C 180,E1 -22719.44,E2 -22719.44} C_VEL
LIN {X 0,Y 227.848,Z 359.14,A -85,B 0,C 180,E1 -22718.823,E2 -22718.823} C_VEL
LIN {X 0,Y 227.026,Z 364.99,A -85,B 0,C 180,E1 -22718.855,E2 -22718.855} C_VEL
LIN {X 0,Y 224.306,Z 401.124,A -85,B 0,C 180,E1 -22719.859,E2 -22719.859} C_VEL
LIN {X 0,Y 221.976,Z 417.234,A -85,B 0,C 180,E1 -22720.549,E2 -22720.549} C_VEL
LIN {X 0,Y 218.828,Z 432.471,A -85,B 0,C 180,E1 -22721.522,E2 -22721.522} C_VEL
LIN {X 0,Y 215.104,Z 446.199,A -85,B 0,C 180,E1 -22722.683,E2 -22722.683} C_VEL
LIN {X 0,Y 210.799,Z 459.654,A -85,B 0,C 180,E1 -22724.21,E2 -22724.21} C_VEL
LIN {X 0,Y 205.972,Z 472.63,A -85,B 0,C 180,E1 -22726.104,E2 -22726.104} C_VEL
LIN {X 0,Y 200.188,Z 485.773,A -85,B 0,C 180,E1 -22728.499,E2 -22728.499} C_VEL
LIN {X 0,Y 194.324,Z 497.949,A -85,B 0,C 180,E1 -22731.402,E2 -22731.402} C_VEL
LIN {X 0,Y 188.575,Z 508.787,A -85,B 0,C 180,E1 -22734.714,E2 -22734.714} C_VEL
LIN {X 0,Y 183.647,Z 517.826,A -85,B 0,C 180,E1 -22738.252,E2 -22738.252} C_VEL
LIN {X 0,Y 179.215,Z 525.325,A -85,B 0,C 180,E1 -22741.929,E2 -22741.929} C_VEL
LIN {X 0,Y 175.218,Z 532.33,A -85,B 0,C 180,E1 -22746.354,E2 -22746.354} C_VEL
LIN {X 0,Y 172.25,Z 537.846,A -85,B 0,C 180,E1 -22750.95,E2 -22750.95} C_VEL
LIN {X 0,Y 170.174,Z 542.021,A -85,B 0,C 180,E1 -22755.653,E2 -22755.653} C_VEL
LIN {X 0,Y 169.122,Z 544.958,A -85,B 0,C 180,E1 -22760.432,E2 -22760.432} C_VEL
LIN {X 0,Y 168.792,Z 546.715,A -85,B 0,C 180,E1 -22765.223,E2 -22765.223} C_VEL
LIN {X 0,Y 168.983,Z 547.321,A -85,B 0,C 180,E1 -22770,E2 -22770} C_VEL
LIN {X 0,Y 168.792,Z 546.698,A -85,B 0,C 180,E1 -22774.777,E2 -22774.777} C_VEL
LIN {X 0,Y 169.122,Z 544.92,A -85,B 0,C 180,E1 -22779.568,E2 -22779.568} C_VEL
LIN {X 0,Y 170.159,Z 541.965,A -85,B 0,C 180,E1 -22784.348,E2 -22784.348} C_VEL
LIN {X 0,Y 172.199,Z 537.774,A -85,B 0,C 180,E1 -22789.056,E2 -22789.056} C_VEL
LIN {X 0,Y 175.194,Z 532.232,A -85,B 0,C 180,E1 -22793.65,E2 -22793.65} C_VEL
LIN {X 0,Y 179.212,Z 525.195,A -85,B 0,C 180,E1 -22798.072,E2 -22798.072} C_VEL
LIN {X 0,Y 183.638,Z 517.68,A -85,B 0,C 180,E1 -22801.75,E2 -22801.75} C_VEL
LIN {X 0,Y 187.803,Z 509.981,A -85,B 0,C 180,E1 -22804.797,E2 -22804.797} C_VEL
LIN {X 0,Y 192.594,Z 501.016,A -85,B 0,C 180,E1 -22807.677,E2 -22807.677} C_VEL
LIN {X 0,Y 197.844,Z 490.458,A -85,B 0,C 180,E1 -22810.412,E2 -22810.412} C_VEL
LIN {X 0,Y 203.138,Z 478.985,A -85,B 0,C 180,E1 -22812.762,E2 -22812.762} C_VEL
LIN {X 0,Y 208.137,Z 466.654,A -85,B 0,C 180,E1 -22814.783,E2 -22814.783} C_VEL
LIN {X 0,Y 212.927,Z 452.84,A -85,B 0,C 180,E1 -22816.563,E2 -22816.563} C_VEL
LIN {X 0,Y 217.034,Z 438.674,A -85,B 0,C 180,E1 -22817.966,E2 -22817.966} C_VEL
LIN {X 0,Y 220.648,Z 423.33,A -85,B 0,C 180,E1 -22819.066,E2 -22819.066} C_VEL
LIN {X 0,Y 223.275,Z 408.058,A -85,B 0,C 180,E1 -22819.837,E2 -22819.837} C_VEL
LIN {X 0,Y 224.925,Z 392.043,A -85,B 0,C 180,E1 -22820.375,E2 -22820.375} C_VEL
LIN {X 0,Y 229.569,Z 326.519,A -85,B 0,C 180,E1 -22822.154,E2 -22822.154} C_VEL
LIN {X 0,Y 224.7,Z 314.661,A -85,B 0,C 180,E1 -22824.398,E2 -22824.398} C_VEL
LIN {X 0,Y 219.009,Z 302.713,A -85,B 0,C 180,E1 -22827.213,E2 -22827.213} C_VEL
LIN {X 0,Y 214.47,Z 293.953,A -85,B 0,C 180,E1 -22829.691,E2 -22829.691} C_VEL
LIN {X 0,Y 210.403,Z 286.923,A -85,B 0,C 180,E1 -22832.119,E2 -22832.119} C_VEL
LIN {X 0,Y 207.363,Z 282.668,A -85,B 0,C 180,E1 -22834.061,E2 -22834.061} C_VEL
LIN {X 0,Y 204.753,Z 279.026,A -85,B 0,C 180,E1 -22835.891,E2 -22835.891} C_VEL
LIN {X 0,Y 201.574,Z 274.757,A -85,B 0,C 180,E1 -22838.371,E2 -22838.371} C_VEL
LIN {X 0,Y 198.815,Z 271.288,A -85,B 0,C 180,E1 -22840.814,E2 -22840.814} C_VEL
LIN {X 0,Y 198.001,Z 269.988,A -85,B 0,C 180,E1 -22841.638,E2 -22841.638} C_VEL
LIN {X 0,Y 195.478,Z 267.428,A -85,B 0,C 180,E1 -22844.314,E2 -22844.314} C_VEL
LIN {X 0,Y 193.957,Z 264.733,A -85,B 0,C 180,E1 -22846.378,E2 -22846.378} C_VEL
LIN {X 0,Y 191.345,Z 262.561,A -85,B 0,C 180,E1 -22850.487,E2 -22850.487} C_VEL
LIN {X 0,Y 189.893,Z 259.149,A -85,B 0,C 180,E1 -22854.691,E2 -22854.691} C_VEL
LIN {X 0,Y 189.068,Z 258.678,A -85,B 0,C 180,E1 -22860,E2 -22860} C_VEL
LIN {X 0,Y 190.035,Z 259.311,A -85,B 0,C 180,E1 -22866.237,E2 -22866.237} C_VEL
LIN {X 0,Y 191.259,Z 262.47,A -85,B 0,C 180,E1 -22869.785,E2 -22869.785} C_VEL
LIN {X 0,Y 193.633,Z 264.575,A -85,B 0,C 180,E1 -22873.646,E2 -22873.646} C_VEL
LIN {X 0,Y 194.252,Z 265.112,A -85,B 0,C 180,E1 -22874.47,E2 -22874.47} C_VEL
LIN {X 0,Y 196.154,Z 268.364,A -85,B 0,C 180,E1 -22876.925,E2 -22876.925} C_VEL
LIN {X 0,Y 198.39,Z 270.531,A -85,B 0,C 180,E1 -22879.196,E2 -22879.196} C_VEL
LIN {X 0,Y 200.753,Z 273.972,A -85,B 0,C 180,E1 -22881.405,E2 -22881.405} C_VEL
LIN {X 0,Y 202.309,Z 275.653,A -85,B 0,C 180,E1 -22882.668,E2 -22882.668} C_VEL
LIN {X 0,Y 205.928,Z 280.631,A -85,B 0,C 180,E1 -22885.395,E2 -22885.395} C_VEL
LIN {X 0,Y 209.553,Z 285.749,A -85,B 0,C 180,E1 -22887.8,E2 -22887.8} C_VEL
LIN {X 0,Y 213.874,Z 291.91,A -85,B 0,C 180,E1 -22890.347,E2 -22890.347} C_VEL
LIN {X 0,Y 220.526,Z 302.667,A -85,B 0,C 180,E1 -22893.829,E2 -22893.829} C_VEL
LIN {X 0,Y 226.546,Z 313.333,A -85,B 0,C 180,E1 -22896.618,E2 -22896.618} C_VEL
LIN {X 0,Y 229.954,Z 319.949,A -85,B 0,C 180,E1 -22898.085,E2 -22898.085} C_VEL
LIN {X 0,Y 224.621,Z 393.212,A -85,B 0,C 180,E1 -22900.107,E2 -22900.107} C_VEL
LIN {X 0,Y 222.514,Z 408.624,A -85,B 0,C 180,E1 -22900.797,E2 -22900.797} C_VEL
LIN {X 0,Y 219.617,Z 423.335,A -85,B 0,C 180,E1 -22901.754,E2 -22901.754} C_VEL
LIN {X 0,Y 215.858,Z 438.233,A -85,B 0,C 180,E1 -22903.094,E2 -22903.094} C_VEL
LIN {X 0,Y 211.602,Z 452.217,A -85,B 0,C 180,E1 -22904.772,E2 -22904.772} C_VEL
LIN {X 0,Y 206.55,Z 465.658,A -85,B 0,C 180,E1 -22906.784,E2 -22906.784} C_VEL
LIN {X 0,Y 201.342,Z 477.857,A -85,B 0,C 180,E1 -22909.121,E2 -22909.121} C_VEL
LIN {X 0,Y 195.928,Z 488.973,A -85,B 0,C 180,E1 -22911.775,E2 -22911.775} C_VEL
LIN {X 0,Y 191.913,Z 496.834,A -85,B 0,C 180,E1 -22914.132,E2 -22914.132} C_VEL
LIN {X 0,Y 187.373,Z 505.05,A -85,B 0,C 180,E1 -22917.054,E2 -22917.054} C_VEL
LIN {X 0,Y 182.717,Z 513.122,A -85,B 0,C 180,E1 -22920.633,E2 -22920.633} C_VEL
LIN {X 0,Y 178.646,Z 519.784,A -85,B 0,C 180,E1 -22924.359,E2 -22924.359} C_VEL
LIN {X 0,Y 175.054,Z 525.937,A -85,B 0,C 180,E1 -22928.819,E2 -22928.819} C_VEL
LIN {X 0,Y 172.227,Z 530.687,A -85,B 0,C 180,E1 -22933.403,E2 -22933.403} C_VEL
LIN {X 0,Y 170.435,Z 534.155,A -85,B 0,C 180,E1 -22938.102,E2 -22938.102} C_VEL
LIN {X 0,Y 169.42,Z 536.442,A -85,B 0,C 180,E1 -22942.851,E2 -22942.851} C_VEL
LIN {X 0,Y 169.01,Z 537.604,A -85,B 0,C 180,E1 -22947.617,E2 -22947.617} C_VEL
LIN {X 0,Y 169.027,Z 537.758,A -85,B 0,C 180,E1 -22950,E2 -22950} C_VEL
LIN {X 0,Y 169.146,Z 537.196,A -85,B 0,C 180,E1 -22954.767,E2 -22954.767} C_VEL
LIN {X 0,Y 169.837,Z 535.522,A -85,B 0,C 180,E1 -22959.527,E2 -22959.527} C_VEL
LIN {X 0,Y 171.197,Z 532.696,A -85,B 0,C 180,E1 -22964.259,E2 -22964.259} C_VEL
LIN {X 0,Y 173.528,Z 528.64,A -85,B 0,C 180,E1 -22968.905,E2 -22968.905} C_VEL
LIN {X 0,Y 176.741,Z 523.259,A -85,B 0,C 180,E1 -22973.43,E2 -22973.43} C_VEL
LIN {X 0,Y 180.817,Z 516.397,A -85,B 0,C 180,E1 -22977.801,E2 -22977.801} C_VEL
LIN {X 0,Y 185.882,Z 507.824,A -85,B 0,C 180,E1 -22981.959,E2 -22981.959} C_VEL
LIN {X 0,Y 191.043,Z 498.702,A -85,B 0,C 180,E1 -22985.408,E2 -22985.408} C_VEL
LIN {X 0,Y 194.997,Z 491.031,A -85,B 0,C 180,E1 -22987.785,E2 -22987.785} C_VEL
LIN {X 0,Y 200.327,Z 480.308,A -85,B 0,C 180,E1 -22990.467,E2 -22990.467} C_VEL
LIN {X 0,Y 205.43,Z 468.602,A -85,B 0,C 180,E1 -22992.838,E2 -22992.838} C_VEL
LIN {X 0,Y 210.455,Z 455.808,A -85,B 0,C 180,E1 -22994.865,E2 -22994.865} C_VEL
LIN {X 0,Y 214.885,Z 442.059,A -85,B 0,C 180,E1 -22996.62,E2 -22996.62} C_VEL
LIN {X 0,Y 218.695,Z 427.91,A -85,B 0,C 180,E1 -22997.999,E2 -22997.999} C_VEL
LIN {X 0,Y 221.932,Z 412.483,A -85,B 0,C 180,E1 -22999.116,E2 -22999.116} C_VEL
LIN {X 0,Y 224.348,Z 397.015,A -85,B 0,C 180,E1 -22999.866,E2 -22999.866} C_VEL
LIN {X 0,Y 226.081,Z 377.476,A -85,B 0,C 180,E1 -23000.472,E2 -23000.472} C_VEL
LIN {X 0,Y 230.171,Z 320.152,A -85,B 0,C 180,E1 -23002.019,E2 -23002.019} C_VEL
LIN {X 0,Y 224.168,Z 308.837,A -85,B 0,C 180,E1 -23004.655,E2 -23004.655} C_VEL
LIN {X 0,Y 218.349,Z 298.897,A -85,B 0,C 180,E1 -23007.478,E2 -23007.478} C_VEL
LIN {X 0,Y 212.877,Z 290.388,A -85,B 0,C 180,E1 -23010.452,E2 -23010.452} C_VEL
LIN {X 0,Y 207.882,Z 283.212,A -85,B 0,C 180,E1 -23013.543,E2 -23013.543} C_VEL
LIN {X 0,Y 204.814,Z 279.067,A -85,B 0,C 180,E1 -23015.684,E2 -23015.684} C_VEL
LIN {X 0,Y 201.626,Z 274.767,A -85,B 0,C 180,E1 -23018.195,E2 -23018.195} C_VEL
LIN {X 0,Y 198.827,Z 271.184,A -85,B 0,C 180,E1 -23020.714,E2 -23020.714} C_VEL
LIN {X 0,Y 198.176,Z 270.094,A -85,B 0,C 180,E1 -23021.387,E2 -23021.387} C_VEL
LIN {X 0,Y 195.606,Z 267.545,A -85,B 0,C 180,E1 -23024.133,E2 -23024.133} C_VEL
LIN {X 0,Y 194.179,Z 264.783,A -85,B 0,C 180,E1 -23026.126,E2 -23026.126} C_VEL
LIN {X 0,Y 191.642,Z 262.881,A -85,B 0,C 180,E1 -23030.101,E2 -23030.101} C_VEL
LIN {X 0,Y 189.962,Z 259.132,A -85,B 0,C 180,E1 -23035.225,E2 -23035.225} C_VEL
LIN {X 0,Y 189.53,Z 258.912,A -85,B 0,C 180,E1 -23042.125,E2 -23042.125} C_VEL
LIN {X 0,Y 190.085,Z 259.391,A -85,B 0,C 180,E1 -23044.971,E2 -23044.971} C_VEL
LIN {X 0,Y 191.882,Z 263.186,A -85,B 0,C 180,E1 -23050.019,E2 -23050.019} C_VEL
LIN {X 0,Y 194.311,Z 265.12,A -85,B 0,C 180,E1 -23053.73,E2 -23053.73} C_VEL
LIN {X 0,Y 196.339,Z 268.457,A -85,B 0,C 180,E1 -23056.373,E2 -23056.373} C_VEL
LIN {X 0,Y 198.488,Z 270.582,A -85,B 0,C 180,E1 -23058.582,E2 -23058.582} C_VEL
LIN {X 0,Y 201.283,Z 274.426,A -85,B 0,C 180,E1 -23061.171,E2 -23061.171} C_VEL
LIN {X 0,Y 202.506,Z 275.885,A -85,B 0,C 180,E1 -23062.174,E2 -23062.174} C_VEL
LIN {X 0,Y 206.213,Z 280.939,A -85,B 0,C 180,E1 -23064.967,E2 -23064.967} C_VEL
LIN {X 0,Y 209.465,Z 285.49,A -85,B 0,C 180,E1 -23067.135,E2 -23067.135} C_VEL
LIN {X 0,Y 211.717,Z 288.978,A -85,B 0,C 180,E1 -23068.535,E2 -23068.535} C_VEL
LIN {X 0,Y 216.478,Z 297.541,A -85,B 0,C 180,E1 -23071.295,E2 -23071.295} C_VEL
LIN {X 0,Y 222.014,Z 308.673,A -85,B 0,C 180,E1 -23074.186,E2 -23074.186} C_VEL
LIN {X 0,Y 226.919,Z 319.613,A -85,B 0,C 180,E1 -23076.529,E2 -23076.529} C_VEL
LIN {X 0,Y 229.73,Z 326.724,A -85,B 0,C 180,E1 -23077.815,E2 -23077.815} C_VEL
LIN {X 0,Y 227.026,Z 364.99,A -85,B 0,C 180,E1 -23078.855,E2 -23078.855} C_VEL
LIN {X 0,Y 226.227,Z 370.842,A -85,B 0,C 180,E1 -23078.888,E2 -23078.888} C_VEL
LIN {X 0,Y 221.249,Z 389.897,A -85,B 0,C 180,E1 -23078.246,E2 -23078.246} C_VEL
LIN {X 0,Y 220.318,Z 395.738,A -85,B 0,C 180,E1 -23078.281,E2 -23078.281} C_VEL
LIN {X 0,Y 218.475,Z 410.928,A -85,B 0,C 180,E1 -23078.843,E2 -23078.843} C_VEL
LIN {X 0,Y 215.662,Z 425.879,A -85,B 0,C 180,E1 -23079.657,E2 -23079.657} C_VEL
LIN {X 0,Y 212.084,Z 440.039,A -85,B 0,C 180,E1 -23080.711,E2 -23080.711} C_VEL
LIN {X 0,Y 208.113,Z 453.098,A -85,B 0,C 180,E1 -23082.019,E2 -23082.019} C_VEL
LIN {X 0,Y 203.364,Z 466.241,A -85,B 0,C 180,E1 -23083.723,E2 -23083.723} C_VEL
LIN {X 0,Y 197.976,Z 479.075,A -85,B 0,C 180,E1 -23085.841,E2 -23085.841} C_VEL
LIN {X 0,Y 192.467,Z 490.503,A -85,B 0,C 180,E1 -23088.211,E2 -23088.211} C_VEL
LIN {X 0,Y 187.014,Z 501.02,A -85,B 0,C 180,E1 -23090.99,E2 -23090.99} C_VEL
LIN {X 0,Y 181.163,Z 511.309,A -85,B 0,C 180,E1 -23094.416,E2 -23094.416} C_VEL
LIN {X 0,Y 176.217,Z 519.875,A -85,B 0,C 180,E1 -23098.1,E2 -23098.1} C_VEL
LIN {X 0,Y 171.76,Z 527,A -85,B 0,C 180,E1 -23101.931,E2 -23101.931} C_VEL
LIN {X 0,Y 167.749,Z 533.621,A -85,B 0,C 180,E1 -23106.547,E2 -23106.547} C_VEL
LIN {X 0,Y 164.829,Z 538.811,A -85,B 0,C 180,E1 -23111.351,E2 -23111.351} C_VEL
LIN {X 0,Y 163.249,Z 541.82,A -85,B 0,C 180,E1 -23115.031,E2 -23115.031} C_VEL
LIN {X 0,Y 162.086,Z 544.757,A -85,B 0,C 180,E1 -23120.012,E2 -23120.012} C_VEL
LIN {X 0,Y 161.705,Z 546.514,A -85,B 0,C 180,E1 -23125.013,E2 -23125.013} C_VEL
LIN {X 0,Y 161.894,Z 547.121,A -85,B 0,C 180,E1 -23130,E2 -23130} C_VEL
LIN {X 0,Y 161.705,Z 546.497,A -85,B 0,C 180,E1 -23134.987,E2 -23134.987} C_VEL
LIN {X 0,Y 162.085,Z 544.718,A -85,B 0,C 180,E1 -23139.988,E2 -23139.988} C_VEL
LIN {X 0,Y 163.233,Z 541.762,A -85,B 0,C 180,E1 -23144.971,E2 -23144.971} C_VEL
LIN {X 0,Y 165.441,Z 537.57,A -85,B 0,C 180,E1 -23149.867,E2 -23149.867} C_VEL
LIN {X 0,Y 168.64,Z 532.028,A -85,B 0,C 180,E1 -23154.629,E2 -23154.629} C_VEL
LIN {X 0,Y 172.92,Z 524.991,A -85,B 0,C 180,E1 -23159.19,E2 -23159.19} C_VEL
LIN {X 0,Y 177.544,Z 517.475,A -85,B 0,C 180,E1 -23162.975,E2 -23162.975} C_VEL
LIN {X 0,Y 182.779,Z 508.415,A -85,B 0,C 180,E1 -23166.582,E2 -23166.582} C_VEL
LIN {X 0,Y 188.766,Z 497.534,A -85,B 0,C 180,E1 -23169.958,E2 -23169.958} C_VEL
LIN {X 0,Y 194.402,Z 486.337,A -85,B 0,C 180,E1 -23172.674,E2 -23172.674} C_VEL
LIN {X 0,Y 200.326,Z 473.539,A -85,B 0,C 180,E1 -23175.072,E2 -23175.072} C_VEL
LIN {X 0,Y 205.329,Z 460.58,A -85,B 0,C 180,E1 -23177.021,E2 -23177.021} C_VEL
LIN {X 0,Y 209.774,Z 447.325,A -85,B 0,C 180,E1 -23178.556,E2 -23178.556} C_VEL
LIN {X 0,Y 213.527,Z 433.949,A -85,B 0,C 180,E1 -23179.745,E2 -23179.745} C_VEL
LIN {X 0,Y 216.831,Z 419.306,A -85,B 0,C 180,E1 -23180.699,E2 -23180.699} C_VEL
LIN {X 0,Y 219.275,Z 404.034,A -85,B 0,C 180,E1 -23181.398,E2 -23181.398} C_VEL
LIN {X 0,Y 221.222,Z 381.831,A -85,B 0,C 180,E1 -23182.062,E2 -23182.062} C_VEL
LIN {X 0,Y 225.122,Z 329.253,A -85,B 0,C 180,E1 -23183.48,E2 -23183.48} C_VEL
LIN {X 0,Y 220.622,Z 318.089,A -85,B 0,C 180,E1 -23185.699,E2 -23185.699} C_VEL
LIN {X 0,Y 215.304,Z 306.698,A -85,B 0,C 180,E1 -23188.515,E2 -23188.515} C_VEL
LIN {X 0,Y 211.071,Z 298.295,A -85,B 0,C 180,E1 -23190.995,E2 -23190.995} C_VEL
LIN {X 0,Y 207.857,Z 292.704,A -85,B 0,C 180,E1 -23193.032,E2 -23193.032} C_VEL
LIN {X 0,Y 205.32,Z 289.023,A -85,B 0,C 180,E1 -23194.736,E2 -23194.736} C_VEL
LIN {X 0,Y 202.727,Z 285.329,A -85,B 0,C 180,E1 -23196.638,E2 -23196.638} C_VEL
LIN {X 0,Y 199.834,Z 281.301,A -85,B 0,C 180,E1 -23199.005,E2 -23199.005} C_VEL
LIN {X 0,Y 196.989,Z 277.475,A -85,B 0,C 180,E1 -23201.675,E2 -23201.675} C_VEL
LIN {X 0,Y 196.091,Z 276.385,A -85,B 0,C 180,E1 -23202.602,E2 -23202.602} C_VEL
LIN {X 0,Y 193.774,Z 273.61,A -85,B 0,C 180,E1 -23205.293,E2 -23205.293} C_VEL
LIN {X 0,Y 192.719,Z 271.633,A -85,B 0,C 180,E1 -23206.825,E2 -23206.825} C_VEL
LIN {X 0,Y 190.168,Z 269.3,A -85,B 0,C 180,E1 -23211.098,E2 -23211.098} C_VEL
LIN {X 0,Y 189.026,Z 266.237,A -85,B 0,C 180,E1 -23214.667,E2 -23214.667} C_VEL
LIN {X 0,Y 188.203,Z 265.724,A -85,B 0,C 180,E1 -23220,E2 -23220} C_VEL
LIN {X 0,Y 189.047,Z 266.304,A -85,B 0,C 180,E1 -23225.868,E2 -23225.868} C_VEL
LIN {X 0,Y 190.268,Z 269.469,A -85,B 0,C 180,E1 -23229.568,E2 -23229.568} C_VEL
LIN {X 0,Y 192.96,Z 271.953,A -85,B 0,C 180,E1 -23233.963,E2 -23233.963} C_VEL
LIN {X 0,Y 194.96,Z 275.325,A -85,B 0,C 180,E1 -23236.627,E2 -23236.627} C_VEL
LIN {X 0,Y 196.839,Z 277.228,A -85,B 0,C 180,E1 -23238.609,E2 -23238.609} C_VEL
LIN {X 0,Y 199.508,Z 281.004,A -85,B 0,C 180,E1 -23241.166,E2 -23241.166} C_VEL
LIN {X 0,Y 200.634,Z 282.38,A -85,B 0,C 180,E1 -23242.121,E2 -23242.121} C_VEL
LIN {X 0,Y 203.998,Z 287.114,A -85,B 0,C 180,E1 -23244.759,E2 -23244.759} C_VEL
LIN {X 0,Y 207.838,Z 292.688,A -85,B 0,C 180,E1 -23247.4,E2 -23247.4} C_VEL
LIN {X 0,Y 212.771,Z 300.234,A -85,B 0,C 180,E1 -23250.384,E2 -23250.384} C_VEL
LIN {X 0,Y 218.06,Z 309.093,A -85,B 0,C 180,E1 -23253.224,E2 -23253.224} C_VEL
LIN {X 0,Y 223.602,Z 319.239,A -85,B 0,C 180,E1 -23255.901,E2 -23255.901} C_VEL
LIN {X 0,Y 225.479,Z 322.986,A -85,B 0,C 180,E1 -23256.757,E2 -23256.757} C_VEL
LIN {X 0,Y 220.15,Z 393.232,A -85,B 0,C 180,E1 -23258.691,E2 -23258.691} C_VEL
LIN {X 0,Y 217.961,Z 408.835,A -85,B 0,C 180,E1 -23259.39,E2 -23259.39} C_VEL
LIN {X 0,Y 214.967,Z 423.543,A -85,B 0,C 180,E1 -23260.346,E2 -23260.346} C_VEL
LIN {X 0,Y 211.419,Z 437.191,A -85,B 0,C 180,E1 -23261.562,E2 -23261.562} C_VEL
LIN {X 0,Y 207.189,Z 450.875,A -85,B 0,C 180,E1 -23263.174,E2 -23263.174} C_VEL
LIN {X 0,Y 201.934,Z 464.623,A -85,B 0,C 180,E1 -23265.19,E2 -23265.19} C_VEL
LIN {X 0,Y 196.492,Z 477.026,A -85,B 0,C 180,E1 -23267.539,E2 -23267.539} C_VEL
LIN {X 0,Y 191.266,Z 487.412,A -85,B 0,C 180,E1 -23269.983,E2 -23269.983} C_VEL
LIN {X 0,Y 187.02,Z 495.375,A -85,B 0,C 180,E1 -23272.277,E2 -23272.277} C_VEL
LIN {X 0,Y 183.035,Z 502.645,A -85,B 0,C 180,E1 -23274.834,E2 -23274.834} C_VEL
LIN {X 0,Y 177.85,Z 511.134,A -85,B 0,C 180,E1 -23278.427,E2 -23278.427} C_VEL
LIN {X 0,Y 173.408,Z 518.192,A -85,B 0,C 180,E1 -23282.22,E2 -23282.22} C_VEL
LIN {X 0,Y 169.241,Z 524.733,A -85,B 0,C 180,E1 -23286.766,E2 -23286.766} C_VEL
LIN {X 0,Y 166.077,Z 529.838,A -85,B 0,C 180,E1 -23291.496,E2 -23291.496} C_VEL
LIN {X 0,Y 164.331,Z 532.776,A -85,B 0,C 180,E1 -23295.132,E2 -23295.132} C_VEL
LIN {X 0,Y 162.832,Z 535.644,A -85,B 0,C 180,E1 -23300.059,E2 -23300.059} C_VEL
LIN {X 0,Y 162.067,Z 537.363,A -85,B 0,C 180,E1 -23305.025,E2 -23305.025} C_VEL
LIN {X 0,Y 161.939,Z 537.958,A -85,B 0,C 180,E1 -23310,E2 -23310} C_VEL
LIN {X 0,Y 162.067,Z 537.397,A -85,B 0,C 180,E1 -23314.975,E2 -23314.975} C_VEL
LIN {X 0,Y 162.825,Z 535.723,A -85,B 0,C 180,E1 -23319.942,E2 -23319.942} C_VEL
LIN {X 0,Y 164.291,Z 532.897,A -85,B 0,C 180,E1 -23324.872,E2 -23324.872} C_VEL
LIN {X 0,Y 166.812,Z 528.84,A -85,B 0,C 180,E1 -23329.697,E2 -23329.697} C_VEL
LIN {X 0,Y 170.221,Z 523.459,A -85,B 0,C 180,E1 -23334.385,E2 -23334.385} C_VEL
LIN {X 0,Y 174.547,Z 516.597,A -85,B 0,C 180,E1 -23338.892,E2 -23338.892} C_VEL
LIN {X 0,Y 179.853,Z 508.024,A -85,B 0,C 180,E1 -23343.165,E2 -23343.165} C_VEL
LIN {X 0,Y 185.257,Z 498.902,A -85,B 0,C 180,E1 -23346.69,E2 -23346.69} C_VEL
LIN {X 0,Y 189.423,Z 491.23,A -85,B 0,C 180,E1 -23349.103,E2 -23349.103} C_VEL
LIN {X 0,Y 194.975,Z 480.506,A -85,B 0,C 180,E1 -23351.823,E2 -23351.823} C_VEL
LIN {X 0,Y 199.772,Z 469.969,A -85,B 0,C 180,E1 -23354.01,E2 -23354.01} C_VEL
LIN {X 0,Y 204.942,Z 457.425,A -85,B 0,C 180,E1 -23356.065,E2 -23356.065} C_VEL
LIN {X 0,Y 209.459,Z 444.258,A -85,B 0,C 180,E1 -23357.806,E2 -23357.806} C_VEL
LIN {X 0,Y 213.471,Z 430.357,A -85,B 0,C 180,E1 -23359.218,E2 -23359.218} C_VEL
LIN {X 0,Y 216.844,Z 415.714,A -85,B 0,C 180,E1 -23360.329,E2 -23360.329} C_VEL
LIN {X 0,Y 219.347,Z 401.052,A -85,B 0,C 180,E1 -23361.128,E2 -23361.128} C_VEL
LIN {X 0,Y 221.092,Z 384.743,A -85,B 0,C 180,E1 -23361.7,E2 -23361.7} C_VEL
LIN {X 0,Y 225.655,Z 323.101,A -85,B 0,C 180,E1 -23363.367,E2 -23363.367} C_VEL
LIN {X 0,Y 219.661,Z 311.754,A -85,B 0,C 180,E1 -23366.19,E2 -23366.19} C_VEL
LIN {X 0,Y 214.051,Z 302.161,A -85,B 0,C 180,E1 -23369.131,E2 -23369.131} C_VEL
LIN {X 0,Y 209.101,Z 294.249,A -85,B 0,C 180,E1 -23372.066,E2 -23372.066} C_VEL
LIN {X 0,Y 205.12,Z 288.656,A -85,B 0,C 180,E1 -23374.707,E2 -23374.707} C_VEL
LIN {X 0,Y 202.707,Z 285.24,A -85,B 0,C 180,E1 -23376.502,E2 -23376.502} C_VEL
LIN {X 0,Y 199.814,Z 281.215,A -85,B 0,C 180,E1 -23378.901,E2 -23378.901} C_VEL
LIN {X 0,Y 197.158,Z 277.65,A -85,B 0,C 180,E1 -23381.422,E2 -23381.422} C_VEL
LIN {X 0,Y 196.456,Z 276.676,A -85,B 0,C 180,E1 -23382.162,E2 -23382.162} C_VEL
LIN {X 0,Y 193.963,Z 273.825,A -85,B 0,C 180,E1 -23385.045,E2 -23385.045} C_VEL
LIN {X 0,Y 192.752,Z 271.639,A -85,B 0,C 180,E1 -23386.827,E2 -23386.827} C_VEL
LIN {X 0,Y 190.355,Z 269.416,A -85,B 0,C 180,E1 -23390.972,E2 -23390.972} C_VEL
LIN {X 0,Y 189.091,Z 266.214,A -85,B 0,C 180,E1 -23395.221,E2 -23395.221} C_VEL
LIN {X 0,Y 188.528,Z 265.835,A -85,B 0,C 180,E1 -23400,E2 -23400} C_VEL
LIN {X 0,Y 189.109,Z 266.291,A -85,B 0,C 180,E1 -23404.529,E2 -23404.529} C_VEL
LIN {X 0,Y 190.832,Z 270.129,A -85,B 0,C 180,E1 -23409.706,E2 -23409.706} C_VEL
LIN {X 0,Y 193.092,Z 272.066,A -85,B 0,C 180,E1 -23413.316,E2 -23413.316} C_VEL
LIN {X 0,Y 195.254,Z 275.548,A -85,B 0,C 180,E1 -23416.198,E2 -23416.198} C_VEL
LIN {X 0,Y 196.984,Z 277.324,A -85,B 0,C 180,E1 -23418.035,E2 -23418.035} C_VEL
LIN {X 0,Y 199.935,Z 281.337,A -85,B 0,C 180,E1 -23420.849,E2 -23420.849} C_VEL
LIN {X 0,Y 204.092,Z 287.124,A -85,B 0,C 180,E1 -23424.189,E2 -23424.189} C_VEL
LIN {X 0,Y 207.755,Z 292.426,A -85,B 0,C 180,E1 -23426.731,E2 -23426.731} C_VEL
LIN {X 0,Y 210.917,Z 297.88,A -85,B 0,C 180,E1 -23428.755,E2 -23428.755} C_VEL
LIN {X 0,Y 215.402,Z 306.71,A -85,B 0,C 180,E1 -23431.4,E2 -23431.4} C_VEL
LIN {X 0,Y 220.541,Z 317.678,A -85,B 0,C 180,E1 -23434.136,E2 -23434.136} C_VEL
LIN {X 0,Y 224.788,Z 328.08,A -85,B 0,C 180,E1 -23436.243,E2 -23436.243} C_VEL
LIN {X 0,Y 225.289,Z 329.471,A -85,B 0,C 180,E1 -23436.488,E2 -23436.488} C_VEL
LIN {X 0,Y 220.318,Z 395.738,A -85,B 0,C 180,E1 -23438.281,E2 -23438.281} C_VEL
LIN {X 0,Y 219.735,Z 399.628,A -85,B 0,C 180,E1 -23438.328,E2 -23438.328} C_VEL
LIN {X 0,Y 217.626,Z 407.241,A -85,B 0,C 180,E1 -23438.225,E2 -23438.225} C_VEL
LIN {X 0,Y 212.844,Z 420.243,A -85,B 0,C 180,E1 -23437.992,E2 -23437.992} C_VEL
LIN {X 0,Y 211.163,Z 425.858,A -85,B 0,C 180,E1 -23438.187,E2 -23438.187} C_VEL
LIN {X 0,Y 207.53,Z 439.844,A -85,B 0,C 180,E1 -23439.227,E2 -23439.227} C_VEL
LIN {X 0,Y 203.406,Z 452.901,A -85,B 0,C 180,E1 -23440.526,E2 -23440.526} C_VEL
LIN {X 0,Y 198.097,Z 467.052,A -85,B 0,C 180,E1 -23442.382,E2 -23442.382} C_VEL
LIN {X 0,Y 192.392,Z 480.013,A -85,B 0,C 180,E1 -23444.577,E2 -23444.577} C_VEL
LIN {X 0,Y 186.206,Z 492.206,A -85,B 0,C 180,E1 -23447.206,E2 -23447.206} C_VEL
LIN {X 0,Y 180.587,Z 502.453,A -85,B 0,C 180,E1 -23450.05,E2 -23450.05} C_VEL
LIN {X 0,Y 174.329,Z 512.866,A -85,B 0,C 180,E1 -23453.735,E2 -23453.735} C_VEL
LIN {X 0,Y 168.784,Z 521.879,A -85,B 0,C 180,E1 -23457.935,E2 -23457.935} C_VEL
LIN {X 0,Y 164.298,Z 528.622,A -85,B 0,C 180,E1 -23461.932,E2 -23461.932} C_VEL
LIN {X 0,Y 160.288,Z 534.858,A -85,B 0,C 180,E1 -23466.759,E2 -23466.759} C_VEL
LIN {X 0,Y 157.443,Z 539.691,A -85,B 0,C 180,E1 -23471.792,E2 -23471.792} C_VEL
LIN {X 0,Y 155.57,Z 543.237,A -85,B 0,C 180,E1 -23476.946,E2 -23476.946} C_VEL
LIN {X 0,Y 154.74,Z 545.578,A -85,B 0,C 180,E1 -23482.169,E2 -23482.169} C_VEL
LIN {X 0,Y 154.662,Z 546.761,A -85,B 0,C 180,E1 -23487.396,E2 -23487.396} C_VEL
LIN {X 0,Y 154.793,Z 546.92,A -85,B 0,C 180,E1 -23490,E2 -23490} C_VEL
LIN {X 0,Y 154.62,Z 546.296,A -85,B 0,C 180,E1 -23495.216,E2 -23495.216} C_VEL
LIN {X 0,Y 155.039,Z 544.515,A -85,B 0,C 180,E1 -23500.447,E2 -23500.447} C_VEL
LIN {X 0,Y 156.334,Z 541.559,A -85,B 0,C 180,E1 -23505.648,E2 -23505.648} C_VEL
LIN {X 0,Y 158.7,Z 537.366,A -85,B 0,C 180,E1 -23510.749,E2 -23510.749} C_VEL
LIN {X 0,Y 162.166,Z 531.824,A -85,B 0,C 180,E1 -23515.682,E2 -23515.682} C_VEL
LIN {X 0,Y 166.708,Z 524.787,A -85,B 0,C 180,E1 -23520.39,E2 -23520.39} C_VEL
LIN {X 0,Y 171.538,Z 517.269,A -85,B 0,C 180,E1 -23524.286,E2 -23524.286} C_VEL
LIN {X 0,Y 177.065,Z 508.21,A -85,B 0,C 180,E1 -23527.967,E2 -23527.967} C_VEL
LIN {X 0,Y 183.332,Z 497.329,A -85,B 0,C 180,E1 -23531.396,E2 -23531.396} C_VEL
LIN {X 0,Y 189.236,Z 486.133,A -85,B 0,C 180,E1 -23534.134,E2 -23534.134} C_VEL
LIN {X 0,Y 195.278,Z 473.515,A -85,B 0,C 180,E1 -23536.521,E2 -23536.521} C_VEL
LIN {X 0,Y 200.543,Z 460.374,A -85,B 0,C 180,E1 -23538.51,E2 -23538.51} C_VEL
LIN {X 0,Y 205.144,Z 447.118,A -85,B 0,C 180,E1 -23540.043,E2 -23540.043} C_VEL
LIN {X 0,Y 209.019,Z 433.741,A -85,B 0,C 180,E1 -23541.227,E2 -23541.227} C_VEL
LIN {X 0,Y 212.409,Z 419.095,A -85,B 0,C 180,E1 -23542.18,E2 -23542.18} C_VEL
LIN {X 0,Y 214.95,Z 403.555,A -85,B 0,C 180,E1 -23542.888,E2 -23542.888} C_VEL
LIN {X 0,Y 216.989,Z 380.96,A -85,B 0,C 180,E1 -23543.555,E2 -23543.555} C_VEL
LIN {X 0,Y 220.734,Z 331.791,A -85,B 0,C 180,E1 -23544.894,E2 -23544.894} C_VEL
LIN {X 0,Y 216.313,Z 320.816,A -85,B 0,C 180,E1 -23547.232,E2 -23547.232} C_VEL
LIN {X 0,Y 211.267,Z 309.68,A -85,B 0,C 180,E1 -23550.136,E2 -23550.136} C_VEL
LIN {X 0,Y 207.424,Z 302.103,A -85,B 0,C 180,E1 -23552.57,E2 -23552.57} C_VEL
LIN {X 0,Y 205.171,Z 298.137,A -85,B 0,C 180,E1 -23554.104,E2 -23554.104} C_VEL
LIN {X 0,Y 200.943,Z 291.867,A -85,B 0,C 180,E1 -23557.238,E2 -23557.238} C_VEL
LIN {X 0,Y 198.003,Z 287.709,A -85,B 0,C 180,E1 -23559.753,E2 -23559.753} C_VEL
LIN {X 0,Y 194.828,Z 283.246,A -85,B 0,C 180,E1 -23562.957,E2 -23562.957} C_VEL
LIN {X 0,Y 192.511,Z 280.48,A -85,B 0,C 180,E1 -23565.734,E2 -23565.734} C_VEL
LIN {X 0,Y 191.494,Z 278.531,A -85,B 0,C 180,E1 -23567.279,E2 -23567.279} C_VEL
LIN {X 0,Y 189.015,Z 276.03,A -85,B 0,C 180,E1 -23571.716,E2 -23571.716} C_VEL
LIN {X 0,Y 188.012,Z 273.198,A -85,B 0,C 180,E1 -23575.176,E2 -23575.176} C_VEL
LIN {X 0,Y 187.337,Z 272.772,A -85,B 0,C 180,E1 -23580,E2 -23580} C_VEL
LIN {X 0,Y 188.092,Z 273.435,A -85,B 0,C 180,E1 -23585.629,E2 -23585.629} C_VEL
LIN {X 0,Y 189.617,Z 276.963,A -85,B 0,C 180,E1 -23590.073,E2 -23590.073} C_VEL
LIN {X 0,Y 191.684,Z 278.785,A -85,B 0,C 180,E1 -23593.45,E2 -23593.45} C_VEL
LIN {X 0,Y 193.772,Z 282.281,A -85,B 0,C 180,E1 -23596.325,E2 -23596.325} C_VEL
LIN {X 0,Y 195.337,Z 283.961,A -85,B 0,C 180,E1 -23598.045,E2 -23598.045} C_VEL
LIN {X 0,Y 198.101,Z 287.84,A -85,B 0,C 180,E1 -23600.779,E2 -23600.779} C_VEL
LIN {X 0,Y 201.876,Z 293.237,A -85,B 0,C 180,E1 -23603.941,E2 -23603.941} C_VEL
LIN {X 0,Y 205.794,Z 299.133,A -85,B 0,C 180,E1 -23606.767,E2 -23606.767} C_VEL
LIN {X 0,Y 210.686,Z 306.865,A -85,B 0,C 180,E1 -23609.844,E2 -23609.844} C_VEL
LIN {X 0,Y 216.477,Z 317.07,A -85,B 0,C 180,E1 -23613.054,E2 -23613.054} C_VEL
LIN {X 0,Y 221.038,Z 325.942,A -85,B 0,C 180,E1 -23615.337,E2 -23615.337} C_VEL
LIN {X 0,Y 216.177,Z 389.602,A -85,B 0,C 180,E1 -23617.108,E2 -23617.108} C_VEL
LIN {X 0,Y 214.171,Z 405.073,A -85,B 0,C 180,E1 -23617.718,E2 -23617.718} C_VEL
LIN {X 0,Y 211.33,Z 419.871,A -85,B 0,C 180,E1 -23618.602,E2 -23618.602} C_VEL
LIN {X 0,Y 207.428,Z 435.074,A -85,B 0,C 180,E1 -23619.86,E2 -23619.86} C_VEL
LIN {X 0,Y 203.466,Z 447.927,A -85,B 0,C 180,E1 -23621.3,E2 -23621.3} C_VEL
LIN {X 0,Y 198.595,Z 460.966,A -85,B 0,C 180,E1 -23623.124,E2 -23623.124} C_VEL
LIN {X 0,Y 193.303,Z 472.975,A -85,B 0,C 180,E1 -23625.218,E2 -23625.218} C_VEL
LIN {X 0,Y 187.818,Z 484.068,A -85,B 0,C 180,E1 -23627.66,E2 -23627.66} C_VEL
LIN {X 0,Y 181.962,Z 494.619,A -85,B 0,C 180,E1 -23630.577,E2 -23630.577} C_VEL
LIN {X 0,Y 177.264,Z 502.849,A -85,B 0,C 180,E1 -23633.509,E2 -23633.509} C_VEL
LIN {X 0,Y 171.822,Z 511.338,A -85,B 0,C 180,E1 -23637.184,E2 -23637.184} C_VEL
LIN {X 0,Y 167.131,Z 518.395,A -85,B 0,C 180,E1 -23641.081,E2 -23641.081} C_VEL
LIN {X 0,Y 162.705,Z 524.936,A -85,B 0,C 180,E1 -23645.774,E2 -23645.774} C_VEL
LIN {X 0,Y 159.331,Z 530.04,A -85,B 0,C 180,E1 -23650.682,E2 -23650.682} C_VEL
LIN {X 0,Y 157.451,Z 532.978,A -85,B 0,C 180,E1 -23654.466,E2 -23654.466} C_VEL
LIN {X 0,Y 155.822,Z 535.846,A -85,B 0,C 180,E1 -23659.607,E2 -23659.607} C_VEL
LIN {X 0,Y 155.005,Z 537.564,A -85,B 0,C 180,E1 -23664.797,E2 -23664.797} C_VEL
LIN {X 0,Y 154.853,Z 538.159,A -85,B 0,C 180,E1 -23670,E2 -23670} C_VEL
LIN {X 0,Y 155.005,Z 537.597,A -85,B 0,C 180,E1 -23675.203,E2 -23675.203} C_VEL
LIN {X 0,Y 155.815,Z 535.924,A -85,B 0,C 180,E1 -23680.394,E2 -23680.394} C_VEL
LIN {X 0,Y 157.415,Z 533.098,A -85,B 0,C 180,E1 -23685.538,E2 -23685.538} C_VEL
LIN {X 0,Y 160.098,Z 529.042,A -85,B 0,C 180,E1 -23690.559,E2 -23690.559} C_VEL
LIN {X 0,Y 163.747,Z 523.66,A -85,B 0,C 180,E1 -23695.416,E2 -23695.416} C_VEL
LIN {X 0,Y 168.326,Z 516.798,A -85,B 0,C 180,E1 -23700.067,E2 -23700.067} C_VEL
LIN {X 0,Y 173.918,Z 508.224,A -85,B 0,C 180,E1 -23704.453,E2 -23704.453} C_VEL
LIN {X 0,Y 179.579,Z 499.102,A -85,B 0,C 180,E1 -23708.052,E2 -23708.052} C_VEL
LIN {X 0,Y 184.858,Z 489.811,A -85,B 0,C 180,E1 -23710.98,E2 -23710.98} C_VEL
LIN {X 0,Y 191.176,Z 477.771,A -85,B 0,C 180,E1 -23713.937,E2 -23713.937} C_VEL
LIN {X 0,Y 196.86,Z 465.472,A -85,B 0,C 180,E1 -23716.296,E2 -23716.296} C_VEL
LIN {X 0,Y 202.04,Z 452.494,A -85,B 0,C 180,E1 -23718.257,E2 -23718.257} C_VEL
LIN {X 0,Y 206.641,Z 438.55,A -85,B 0,C 180,E1 -23719.925,E2 -23719.925} C_VEL
LIN {X 0,Y 210.635,Z 423.759,A -85,B 0,C 180,E1 -23721.252,E2 -23721.252} C_VEL
LIN {X 0,Y 213.799,Z 408.359,A -85,B 0,C 180,E1 -23722.258,E2 -23722.258} C_VEL
LIN {X 0,Y 215.954,Z 393.593,A -85,B 0,C 180,E1 -23722.904,E2 -23722.904} C_VEL
LIN {X 0,Y 221.321,Z 326.245,A -85,B 0,C 180,E1 -23724.74,E2 -23724.74} C_VEL
LIN {X 0,Y 215.059,Z 314.279,A -85,B 0,C 180,E1 -23727.924,E2 -23727.924} C_VEL
LIN {X 0,Y 209.521,Z 304.792,A -85,B 0,C 180,E1 -23731.103,E2 -23731.103} C_VEL
LIN {X 0,Y 205.7,Z 298.838,A -85,B 0,C 180,E1 -23733.566,E2 -23733.566} C_VEL
LIN {X 0,Y 201.389,Z 292.322,A -85,B 0,C 180,E1 -23736.748,E2 -23736.748} C_VEL
LIN {X 0,Y 198.167,Z 287.807,A -85,B 0,C 180,E1 -23739.499,E2 -23739.499} C_VEL
LIN {X 0,Y 195.467,Z 283.997,A -85,B 0,C 180,E1 -23742.204,E2 -23742.204} C_VEL
LIN {X 0,Y 192.402,Z 280.134,A -85,B 0,C 180,E1 -23745.928,E2 -23745.928} C_VEL
LIN {X 0,Y 191.545,Z 278.479,A -85,B 0,C 180,E1 -23747.282,E2 -23747.282} C_VEL
LIN {X 0,Y 189.369,Z 276.438,A -85,B 0,C 180,E1 -23751.194,E2 -23751.194} C_VEL
LIN {X 0,Y 188.106,Z 273.205,A -85,B 0,C 180,E1 -23755.714,E2 -23755.714} C_VEL
LIN {X 0,Y 187.666,Z 272.858,A -85,B 0,C 180,E1 -23760,E2 -23760} C_VEL
LIN {X 0,Y 188.196,Z 273.459,A -85,B 0,C 180,E1 -23764.417,E2 -23764.417} C_VEL
LIN {X 0,Y 189.97,Z 277.254,A -85,B 0,C 180,E1 -23769.751,E2 -23769.751} C_VEL
LIN {X 0,Y 191.762,Z 278.786,A -85,B 0,C 180,E1 -23772.703,E2 -23772.703} C_VEL
LIN {X 0,Y 194.067,Z 282.489,A -85,B 0,C 180,E1 -23775.894,E2 -23775.894} C_VEL
LIN {X 0,Y 195.465,Z 284.03,A -85,B 0,C 180,E1 -23777.445,E2 -23777.445} C_VEL
LIN {X 0,Y 199.051,Z 289.047,A -85,B 0,C 180,E1 -23780.946,E2 -23780.946} C_VEL
LIN {X 0,Y 202.309,Z 293.791,A -85,B 0,C 180,E1 -23783.63,E2 -23783.63} C_VEL
LIN {X 0,Y 205.886,Z 299.125,A -85,B 0,C 180,E1 -23786.207,E2 -23786.207} C_VEL
LIN {X 0,Y 210.399,Z 307.677,A -85,B 0,C 180,E1 -23789.175,E2 -23789.175} C_VEL
LIN {X 0,Y 215.539,Z 318.772,A -85,B 0,C 180,E1 -23792.202,E2 -23792.202} C_VEL
LIN {X 0,Y 219.622,Z 328.571,A -85,B 0,C 180,E1 -23794.402,E2 -23794.402} C_VEL
LIN {X 0,Y 220.91,Z 331.999,A -85,B 0,C 180,E1 -23795.074,E2 -23795.074} C_VEL
LIN {X 0,Y 215.434,Z 401.132,A -85,B 0,C 180,E1 -23796.973,E2 -23796.973} C_VEL
LIN {X 0,Y 213.013,Z 416.851,A -85,B 0,C 180,E1 -23797.644,E2 -23797.644} C_VEL
LIN {X 0,Y 211.163,Z 425.858,A -85,B 0,C 180,E1 -23798.187,E2 -23798.187} C_VEL
LIN {X 0,Y 209.35,Z 431.457,A -85,B 0,C 180,E1 -23798.4,E2 -23798.4} C_VEL
LIN {X 0,Y 201.355,Z 447.396,A -85,B 0,C 180,E1 -23798.623,E2 -23798.623} C_VEL
LIN {X 0,Y 198.918,Z 452.626,A -85,B 0,C 180,E1 -23798.97,E2 -23798.97} C_VEL
LIN {X 0,Y 198.248,Z 454.342,A -85,B 0,C 180,E1 -23799.161,E2 -23799.161} C_VEL
LIN {X 0,Y 192.939,Z 467.809,A -85,B 0,C 180,E1 -23800.97,E2 -23800.97} C_VEL
LIN {X 0,Y 187.464,Z 479.815,A -85,B 0,C 180,E1 -23803.027,E2 -23803.027} C_VEL
LIN {X 0,Y 181.021,Z 492.006,A -85,B 0,C 180,E1 -23805.668,E2 -23805.668} C_VEL
LIN {X 0,Y 175.174,Z 502.254,A -85,B 0,C 180,E1 -23808.55,E2 -23808.55} C_VEL
LIN {X 0,Y 168.637,Z 512.641,A -85,B 0,C 180,E1 -23812.288,E2 -23812.288} C_VEL
LIN {X 0,Y 163.478,Z 520.597,A -85,B 0,C 180,E1 -23816.023,E2 -23816.023} C_VEL
LIN {X 0,Y 157.998,Z 528.421,A -85,B 0,C 180,E1 -23820.706,E2 -23820.706} C_VEL
LIN {X 0,Y 153.737,Z 534.656,A -85,B 0,C 180,E1 -23825.706,E2 -23825.706} C_VEL
LIN {X 0,Y 150.634,Z 539.488,A -85,B 0,C 180,E1 -23830.938,E2 -23830.938} C_VEL
LIN {X 0,Y 148.595,Z 543.035,A -85,B 0,C 180,E1 -23836.321,E2 -23836.321} C_VEL
LIN {X 0,Y 147.688,Z 545.377,A -85,B 0,C 180,E1 -23841.793,E2 -23841.793} C_VEL
LIN {X 0,Y 147.564,Z 546.56,A -85,B 0,C 180,E1 -23847.27,E2 -23847.27} C_VEL
LIN {X 0,Y 147.716,Z 546.72,A -85,B 0,C 180,E1 -23850,E2 -23850} C_VEL
LIN {X 0,Y 147.533,Z 546.094,A -85,B 0,C 180,E1 -23855.467,E2 -23855.467} C_VEL
LIN {X 0,Y 148.014,Z 544.312,A -85,B 0,C 180,E1 -23860.948,E2 -23860.948} C_VEL
LIN {X 0,Y 149.46,Z 541.356,A -85,B 0,C 180,E1 -23866.387,E2 -23866.387} C_VEL
LIN {X 0,Y 152.003,Z 537.161,A -85,B 0,C 180,E1 -23871.708,E2 -23871.708} C_VEL
LIN {X 0,Y 155.737,Z 531.62,A -85,B 0,C 180,E1 -23876.825,E2 -23876.825} C_VEL
LIN {X 0,Y 160.576,Z 524.583,A -85,B 0,C 180,E1 -23881.682,E2 -23881.682} C_VEL
LIN {X 0,Y 165.637,Z 517.063,A -85,B 0,C 180,E1 -23885.69,E2 -23885.69} C_VEL
LIN {X 0,Y 171.46,Z 508.005,A -85,B 0,C 180,E1 -23889.444,E2 -23889.444} C_VEL
LIN {X 0,Y 178.024,Z 497.124,A -85,B 0,C 180,E1 -23892.92,E2 -23892.92} C_VEL
LIN {X 0,Y 184.19,Z 485.928,A -85,B 0,C 180,E1 -23895.677,E2 -23895.677} C_VEL
LIN {X 0,Y 190.341,Z 473.526,A -85,B 0,C 180,E1 -23898.039,E2 -23898.039} C_VEL
LIN {X 0,Y 195.888,Z 460.168,A -85,B 0,C 180,E1 -23900.073,E2 -23900.073} C_VEL
LIN {X 0,Y 200.643,Z 446.911,A -85,B 0,C 180,E1 -23901.602,E2 -23901.602} C_VEL
LIN {X 0,Y 204.649,Z 433.533,A -85,B 0,C 180,E1 -23902.776,E2 -23902.776} C_VEL
LIN {X 0,Y 208.132,Z 418.885,A -85,B 0,C 180,E1 -23903.723,E2 -23903.723} C_VEL
LIN {X 0,Y 210.624,Z 404.16,A -85,B 0,C 180,E1 -23904.399,E2 -23904.399} C_VEL
LIN {X 0,Y 212.616,Z 383.501,A -85,B 0,C 180,E1 -23905.022,E2 -23905.022} C_VEL
LIN {X 0,Y 216.478,Z 334.411,A -85,B 0,C 180,E1 -23906.363,E2 -23906.363} C_VEL
LIN {X 0,Y 212.356,Z 324.018,A -85,B 0,C 180,E1 -23908.711,E2 -23908.711} C_VEL
LIN {X 0,Y 207.328,Z 312.657,A -85,B 0,C 180,E1 -23911.858,E2 -23911.858} C_VEL
LIN {X 0,Y 203.529,Z 305.165,A -85,B 0,C 180,E1 -23914.498,E2 -23914.498} C_VEL
LIN {X 0,Y 200.563,Z 300.599,A -85,B 0,C 180,E1 -23916.715,E2 -23916.715} C_VEL
LIN {X 0,Y 198.288,Z 297.212,A -85,B 0,C 180,E1 -23918.599,E2 -23918.599} C_VEL
LIN {X 0,Y 196.371,Z 294.304,A -85,B 0,C 180,E1 -23920.362,E2 -23920.362} C_VEL
LIN {X 0,Y 193.298,Z 289.906,A -85,B 0,C 180,E1 -23923.612,E2 -23923.612} C_VEL
LIN {X 0,Y 190.919,Z 286.694,A -85,B 0,C 180,E1 -23926.699,E2 -23926.699} C_VEL
LIN {X 0,Y 190.284,Z 285.397,A -85,B 0,C 180,E1 -23927.739,E2 -23927.739} C_VEL
LIN {X 0,Y 187.953,Z 282.9,A -85,B 0,C 180,E1 -23932.153,E2 -23932.153} C_VEL
LIN {X 0,Y 187.078,Z 280.218,A -85,B 0,C 180,E1 -23935.421,E2 -23935.421} C_VEL
LIN {X 0,Y 186.472,Z 279.819,A -85,B 0,C 180,E1 -23940,E2 -23940} C_VEL
LIN {X 0,Y 187.119,Z 280.411,A -85,B 0,C 180,E1 -23945.253,E2 -23945.253} C_VEL
LIN {X 0,Y 188.527,Z 283.851,A -85,B 0,C 180,E1 -23949.657,E2 -23949.657} C_VEL
LIN {X 0,Y 190.422,Z 285.631,A -85,B 0,C 180,E1 -23952.93,E2 -23952.93} C_VEL
LIN {X 0,Y 192.589,Z 289.24,A -85,B 0,C 180,E1 -23956.02,E2 -23956.02} C_VEL
LIN {X 0,Y 193.909,Z 290.791,A -85,B 0,C 180,E1 -23957.535,E2 -23957.535} C_VEL
LIN {X 0,Y 197.346,Z 295.773,A -85,B 0,C 180,E1 -23960.999,E2 -23960.999} C_VEL
LIN {X 0,Y 200.015,Z 299.704,A -85,B 0,C 180,E1 -23963.285,E2 -23963.285} C_VEL
LIN {X 0,Y 204.319,Z 306.339,A -85,B 0,C 180,E1 -23966.493,E2 -23966.493} C_VEL
LIN {X 0,Y 209.187,Z 314.639,A -85,B 0,C 180,E1 -23969.65,E2 -23969.65} C_VEL
LIN {X 0,Y 214.43,Z 324.349,A -85,B 0,C 180,E1 -23972.645,E2 -23972.645} C_VEL
LIN {X 0,Y 216.829,Z 329.144,A -85,B 0,C 180,E1 -23973.911,E2 -23973.911} C_VEL
LIN {X 0,Y 211.573,Z 393.701,A -85,B 0,C 180,E1 -23975.694,E2 -23975.694} C_VEL
LIN {X 0,Y 209.252,Z 409.257,A -85,B 0,C 180,E1 -23976.389,E2 -23976.389} C_VEL
LIN {X 0,Y 206.065,Z 423.96,A -85,B 0,C 180,E1 -23977.338,E2 -23977.338} C_VEL
LIN {X 0,Y 202.01,Z 438.538,A -85,B 0,C 180,E1 -23978.645,E2 -23978.645} C_VEL
LIN {X 0,Y 197.149,Z 452.928,A -85,B 0,C 180,E1 -23980.388,E2 -23980.388} C_VEL
LIN {X 0,Y 191.578,Z 466.273,A -85,B 0,C 180,E1 -23982.416,E2 -23982.416} C_VEL
LIN {X 0,Y 185.732,Z 478.47,A -85,B 0,C 180,E1 -23984.808,E2 -23984.808} C_VEL
LIN {X 0,Y 179.636,Z 489.585,A -85,B 0,C 180,E1 -23987.556,E2 -23987.556} C_VEL
LIN {X 0,Y 174.973,Z 497.449,A -85,B 0,C 180,E1 -23990.011,E2 -23990.011} C_VEL
LIN {X 0,Y 169.836,Z 505.661,A -85,B 0,C 180,E1 -23993.129,E2 -23993.129} C_VEL
LIN {X 0,Y 164.379,Z 513.734,A -85,B 0,C 180,E1 -23996.968,E2 -23996.968} C_VEL
LIN {X 0,Y 159.619,Z 520.394,A -85,B 0,C 180,E1 -24001.032,E2 -24001.032} C_VEL
LIN {X 0,Y 155.228,Z 526.548,A -85,B 0,C 180,E1 -24005.954,E2 -24005.954} C_VEL
LIN {X 0,Y 151.833,Z 531.295,A -85,B 0,C 180,E1 -24011.095,E2 -24011.095} C_VEL
LIN {X 0,Y 149.588,Z 534.762,A -85,B 0,C 180,E1 -24016.414,E2 -24016.414} C_VEL
LIN {X 0,Y 148.275,Z 537.047,A -85,B 0,C 180,E1 -24021.825,E2 -24021.825} C_VEL
LIN {X 0,Y 147.756,Z 538.206,A -85,B 0,C 180,E1 -24027.274,E2 -24027.274} C_VEL
LIN {X 0,Y 147.766,Z 538.359,A -85,B 0,C 180,E1 -24030,E2 -24030} C_VEL
LIN {X 0,Y 147.937,Z 537.798,A -85,B 0,C 180,E1 -24035.452,E2 -24035.452} C_VEL
LIN {X 0,Y 148.83,Z 536.125,A -85,B 0,C 180,E1 -24040.888,E2 -24040.888} C_VEL
LIN {X 0,Y 150.568,Z 533.298,A -85,B 0,C 180,E1 -24046.263,E2 -24046.263} C_VEL
LIN {X 0,Y 153.432,Z 529.243,A -85,B 0,C 180,E1 -24051.496,E2 -24051.496} C_VEL
LIN {X 0,Y 157.613,Z 523.394,A -85,B 0,C 180,E1 -24056.899,E2 -24056.899} C_VEL
LIN {X 0,Y 162.201,Z 516.998,A -85,B 0,C 180,E1 -24061.328,E2 -24061.328} C_VEL
LIN {X 0,Y 168.081,Z 508.424,A -85,B 0,C 180,E1 -24065.829,E2 -24065.829} C_VEL
LIN {X 0,Y 173.169,Z 500.71,A -85,B 0,C 180,E1 -24068.98,E2 -24068.98} C_VEL
LIN {X 0,Y 177.563,Z 493.354,A -85,B 0,C 180,E1 -24071.475,E2 -24071.475} C_VEL
LIN {X 0,Y 183.584,Z 482.846,A -85,B 0,C 180,E1 -24074.317,E2 -24074.317} C_VEL
LIN {X 0,Y 189.27,Z 471.532,A -85,B 0,C 180,E1 -24076.778,E2 -24076.778} C_VEL
LIN {X 0,Y 194.815,Z 459.228,A -85,B 0,C 180,E1 -24078.855,E2 -24078.855} C_VEL
LIN {X 0,Y 200.129,Z 444.865,A -85,B 0,C 180,E1 -24080.794,E2 -24080.794} C_VEL
LIN {X 0,Y 204.486,Z 430.744,A -85,B 0,C 180,E1 -24082.229,E2 -24082.229} C_VEL
LIN {X 0,Y 208.064,Z 416.096,A -85,B 0,C 180,E1 -24083.342,E2 -24083.342} C_VEL
LIN {X 0,Y 210.843,Z 400.695,A -85,B 0,C 180,E1 -24084.16,E2 -24084.16} C_VEL
LIN {X 0,Y 212.642,Z 384.757,A -85,B 0,C 180,E1 -24084.702,E2 -24084.702} C_VEL
LIN {X 0,Y 217.041,Z 329.346,A -85,B 0,C 180,E1 -24086.2,E2 -24086.2} C_VEL
LIN {X 0,Y 211.465,Z 318.482,A -85,B 0,C 180,E1 -24089.248,E2 -24089.248} C_VEL
LIN {X 0,Y 205.928,Z 308.8,A -85,B 0,C 180,E1 -24092.682,E2 -24092.682} C_VEL
LIN {X 0,Y 201.311,Z 301.567,A -85,B 0,C 180,E1 -24095.987,E2 -24095.987} C_VEL
LIN {X 0,Y 198.759,Z 297.788,A -85,B 0,C 180,E1 -24098.069,E2 -24098.069} C_VEL
LIN {X 0,Y 196.377,Z 294.236,A -85,B 0,C 180,E1 -24100.26,E2 -24100.26} C_VEL
LIN {X 0,Y 193.471,Z 290.046,A -85,B 0,C 180,E1 -24103.377,E2 -24103.377} C_VEL
LIN {X 0,Y 191.045,Z 286.761,A -85,B 0,C 180,E1 -24106.572,E2 -24106.572} C_VEL
LIN {X 0,Y 190.429,Z 285.435,A -85,B 0,C 180,E1 -24107.613,E2 -24107.613} C_VEL
LIN {X 0,Y 188.284,Z 283.27,A -85,B 0,C 180,E1 -24111.683,E2 -24111.683} C_VEL
LIN {X 0,Y 187.237,Z 280.298,A -85,B 0,C 180,E1 -24115.694,E2 -24115.694} C_VEL
LIN {X 0,Y 186.8,Z 279.906,A -85,B 0,C 180,E1 -24120,E2 -24120} C_VEL
LIN {X 0,Y 187.264,Z 280.506,A -85,B 0,C 180,E1 -24124.17,E2 -24124.17} C_VEL
LIN {X 0,Y 189.023,Z 284.302,A -85,B 0,C 180,E1 -24129.631,E2 -24129.631} C_VEL
LIN {X 0,Y 190.623,Z 285.868,A -85,B 0,C 180,E1 -24132.374,E2 -24132.374} C_VEL
LIN {X 0,Y 192.991,Z 289.545,A -85,B 0,C 180,E1 -24135.714,E2 -24135.714} C_VEL
LIN {X 0,Y 194.079,Z 290.897,A -85,B 0,C 180,E1 -24136.973,E2 -24136.973} C_VEL
LIN {X 0,Y 197.36,Z 295.615,A -85,B 0,C 180,E1 -24140.316,E2 -24140.316} C_VEL
LIN {X 0,Y 200.425,Z 300.252,A -85,B 0,C 180,E1 -24142.962,E2 -24142.962} C_VEL
LIN {X 0,Y 203.741,Z 305.361,A -85,B 0,C 180,E1 -24145.466,E2 -24145.466} C_VEL
LIN {X 0,Y 207.856,Z 313.629,A -85,B 0,C 180,E1 -24148.328,E2 -24148.328} C_VEL
LIN {X 0,Y 212.619,Z 324.367,A -85,B 0,C 180,E1 -24151.296,E2 -24151.296} C_VEL
LIN {X 0,Y 216.479,Z 334.028,A -85,B 0,C 180,E1 -24153.498,E2 -24153.498} C_VEL
LIN {X 0,Y 216.66,Z 335.364,A -85,B 0,C 180,E1 -24153.647,E2 -24153.647} C_VEL
LIN {X 0,Y 211.249,Z 400.923,A -85,B 0,C 180,E1 -24155.435,E2 -24155.435} C_VEL
LIN {X 0,Y 208.756,Z 416.659,A -85,B 0,C 180,E1 -24156.102,E2 -24156.102} C_VEL
LIN {X 0,Y 205.319,Z 431.889,A -85,B 0,C 180,E1 -24157.064,E2 -24157.064} C_VEL
LIN {X 0,Y 201.276,Z 445.614,A -85,B 0,C 180,E1 -24158.222,E2 -24158.222} C_VEL
LIN {X 0,Y 198.248,Z 454.342,A -85,B 0,C 180,E1 -24159.161,E2 -24159.161} C_VEL
LIN {X 0,Y 195.928,Z 459.541,A -85,B 0,C 180,E1 -24159.665,E2 -24159.665} C_VEL
LIN {X 0,Y 186.188,Z 474.108,A -85,B 0,C 180,E1 -24160.65,E2 -24160.65} C_VEL
LIN {X 0,Y 183.161,Z 478.796,A -85,B 0,C 180,E1 -24161.256,E2 -24161.256} C_VEL
LIN {X 0,Y 182.3,Z 480.328,A -85,B 0,C 180,E1 -24161.535,E2 -24161.535} C_VEL
LIN {X 0,Y 175.977,Z 491.807,A -85,B 0,C 180,E1 -24164.04,E2 -24164.04} C_VEL
LIN {X 0,Y 169.872,Z 502.053,A -85,B 0,C 180,E1 -24166.951,E2 -24166.951} C_VEL
LIN {X 0,Y 163.197,Z 512.185,A -85,B 0,C 180,E1 -24170.638,E2 -24170.638} C_VEL
LIN {X 0,Y 157.59,Z 520.396,A -85,B 0,C 180,E1 -24174.568,E2 -24174.568} C_VEL
LIN {X 0,Y 151.787,Z 528.219,A -85,B 0,C 180,E1 -24179.382,E2 -24179.382} C_VEL
LIN {X 0,Y 147.231,Z 534.455,A -85,B 0,C 180,E1 -24184.558,E2 -24184.558} C_VEL
LIN {X 0,Y 143.869,Z 539.286,A -85,B 0,C 180,E1 -24190.005,E2 -24190.005} C_VEL
LIN {X 0,Y 141.641,Z 542.832,A -85,B 0,C 180,E1 -24195.636,E2 -24195.636} C_VEL
LIN {X 0,Y 140.629,Z 545.176,A -85,B 0,C 180,E1 -24201.378,E2 -24201.378} C_VEL
LIN {X 0,Y 140.48,Z 546.36,A -85,B 0,C 180,E1 -24207.132,E2 -24207.132} C_VEL
LIN {X 0,Y 140.568,Z 546.485,A -85,B 0,C 180,E1 -24210.644,E2 -24210.644} C_VEL
LIN {X 0,Y 140.441,Z 545.892,A -85,B 0,C 180,E1 -24215.744,E2 -24215.744} C_VEL
LIN {X 0,Y 141.011,Z 544.109,A -85,B 0,C 180,E1 -24221.499,E2 -24221.499} C_VEL
LIN {X 0,Y 142.614,Z 541.153,A -85,B 0,C 180,E1 -24227.198,E2 -24227.198} C_VEL
LIN {X 0,Y 145.342,Z 536.957,A -85,B 0,C 180,E1 -24232.757,E2 -24232.757} C_VEL
LIN {X 0,Y 149.365,Z 531.416,A -85,B 0,C 180,E1 -24238.068,E2 -24238.068} C_VEL
LIN {X 0,Y 154.527,Z 524.379,A -85,B 0,C 180,E1 -24243.076,E2 -24243.076} C_VEL
LIN {X 0,Y 159.865,Z 516.858,A -85,B 0,C 180,E1 -24247.19,E2 -24247.19} C_VEL
LIN {X 0,Y 165.984,Z 507.8,A -85,B 0,C 180,E1 -24251.017,E2 -24251.017} C_VEL
LIN {X 0,Y 172.867,Z 496.919,A -85,B 0,C 180,E1 -24254.531,E2 -24254.531} C_VEL
LIN {X 0,Y 179.29,Z 485.724,A -85,B 0,C 180,E1 -24257.304,E2 -24257.304} C_VEL
LIN {X 0,Y 185.885,Z 472.779,A -85,B 0,C 180,E1 -24259.777,E2 -24259.777} C_VEL
LIN {X 0,Y 191.39,Z 459.962,A -85,B 0,C 180,E1 -24261.71,E2 -24261.71} C_VEL
LIN {X 0,Y 196.302,Z 446.705,A -85,B 0,C 180,E1 -24263.23,E2 -24263.23} C_VEL
LIN {X 0,Y 200.428,Z 433.325,A -85,B 0,C 180,E1 -24264.395,E2 -24264.395} C_VEL
LIN {X 0,Y 204.013,Z 418.675,A -85,B 0,C 180,E1 -24265.33,E2 -24265.33} C_VEL
LIN {X 0,Y 206.696,Z 402.985,A -85,B 0,C 180,E1 -24266.04,E2 -24266.04} C_VEL
LIN {X 0,Y 208.9,Z 379.965,A -85,B 0,C 180,E1 -24266.709,E2 -24266.709} C_VEL
LIN {X 0,Y 212.367,Z 337.064,A -85,B 0,C 180,E1 -24267.889,E2 -24267.889} C_VEL
LIN {X 0,Y 208.259,Z 326.579,A -85,B 0,C 180,E1 -24270.427,E2 -24270.427} C_VEL
LIN {X 0,Y 204.001,Z 316.784,A -85,B 0,C 180,E1 -24273.324,E2 -24273.324} C_VEL
LIN {X 0,Y 200.733,Z 310.282,A -85,B 0,C 180,E1 -24275.771,E2 -24275.771} C_VEL
LIN {X 0,Y 197.308,Z 304.769,A -85,B 0,C 180,E1 -24278.586,E2 -24278.586} C_VEL
LIN {X 0,Y 194.7,Z 300.806,A -85,B 0,C 180,E1 -24281.043,E2 -24281.043} C_VEL
LIN {X 0,Y 192.016,Z 296.739,A -85,B 0,C 180,E1 -24284.023,E2 -24284.023} C_VEL
LIN {X 0,Y 189.774,Z 293.728,A -85,B 0,C 180,E1 -24287.026,E2 -24287.026} C_VEL
LIN {X 0,Y 189.084,Z 292.288,A -85,B 0,C 180,E1 -24288.204,E2 -24288.204} C_VEL
LIN {X 0,Y 186.842,Z 289.628,A -85,B 0,C 180,E1 -24292.775,E2 -24292.775} C_VEL
LIN {X 0,Y 186.145,Z 287.255,A -85,B 0,C 180,E1 -24295.67,E2 -24295.67} C_VEL
LIN {X 0,Y 185.607,Z 286.867,A -85,B 0,C 180,E1 -24300,E2 -24300} C_VEL
LIN {X 0,Y 186.156,Z 287.373,A -85,B 0,C 180,E1 -24304.873,E2 -24304.873} C_VEL
LIN {X 0,Y 187.537,Z 290.851,A -85,B 0,C 180,E1 -24309.437,E2 -24309.437} C_VEL
LIN {X 0,Y 189.226,Z 292.572,A -85,B 0,C 180,E1 -24312.489,E2 -24312.489} C_VEL
LIN {X 0,Y 191.521,Z 296.276,A -85,B 0,C 180,E1 -24315.839,E2 -24315.839} C_VEL
LIN {X 0,Y 192.58,Z 297.723,A -85,B 0,C 180,E1 -24317.112,E2 -24317.112} C_VEL
LIN {X 0,Y 195.736,Z 302.432,A -85,B 0,C 180,E1 -24320.424,E2 -24320.424} C_VEL
LIN {X 0,Y 198.175,Z 306.227,A -85,B 0,C 180,E1 -24322.617,E2 -24322.617} C_VEL
LIN {X 0,Y 202.188,Z 312.627,A -85,B 0,C 180,E1 -24325.755,E2 -24325.755} C_VEL
LIN {X 0,Y 207.063,Z 321.26,A -85,B 0,C 180,E1 -24329.061,E2 -24329.061} C_VEL
LIN {X 0,Y 211.844,Z 330.547,A -85,B 0,C 180,E1 -24331.92,E2 -24331.92} C_VEL
LIN {X 0,Y 212.744,Z 332.428,A -85,B 0,C 180,E1 -24332.427,E2 -24332.427} C_VEL
LIN {X 0,Y 207.491,Z 394.157,A -85,B 0,C 180,E1 -24334.115,E2 -24334.115} C_VEL
LIN {X 0,Y 205.12,Z 409.468,A -85,B 0,C 180,E1 -24334.793,E2 -24334.793} C_VEL
LIN {X 0,Y 201.843,Z 424.169,A -85,B 0,C 180,E1 -24335.738,E2 -24335.738} C_VEL
LIN {X 0,Y 197.662,Z 438.745,A -85,B 0,C 180,E1 -24337.041,E2 -24337.041} C_VEL
LIN {X 0,Y 193.093,Z 451.911,A -85,B 0,C 180,E1 -24338.62,E2 -24338.62} C_VEL
LIN {X 0,Y 187.456,Z 465.237,A -85,B 0,C 180,E1 -24340.607,E2 -24340.607} C_VEL
LIN {X 0,Y 181.842,Z 476.577,A -85,B 0,C 180,E1 -24342.751,E2 -24342.751} C_VEL
LIN {X 0,Y 175.463,Z 488.025,A -85,B 0,C 180,E1 -24345.498,E2 -24345.498} C_VEL
LIN {X 0,Y 169.555,Z 497.653,A -85,B 0,C 180,E1 -24348.457,E2 -24348.457} C_VEL
LIN {X 0,Y 164.203,Z 505.864,A -85,B 0,C 180,E1 -24351.64,E2 -24351.64} C_VEL
LIN {X 0,Y 158.447,Z 513.937,A -85,B 0,C 180,E1 -24355.562,E2 -24355.562} C_VEL
LIN {X 0,Y 153.432,Z 520.596,A -85,B 0,C 180,E1 -24359.745,E2 -24359.745} C_VEL
LIN {X 0,Y 148.725,Z 526.752,A -85,B 0,C 180,E1 -24364.831,E2 -24364.831} C_VEL
LIN {X 0,Y 145.102,Z 531.498,A -85,B 0,C 180,E1 -24370.182,E2 -24370.182} C_VEL
LIN {X 0,Y 142.667,Z 534.964,A -85,B 0,C 180,E1 -24375.741,E2 -24375.741} C_VEL
LIN {X 0,Y 141.252,Z 537.248,A -85,B 0,C 180,E1 -24381.416,E2 -24381.416} C_VEL
LIN {X 0,Y 140.678,Z 538.407,A -85,B 0,C 180,E1 -24387.136,E2 -24387.136} C_VEL
LIN {X 0,Y 140.653,Z 538.46,A -85,B 0,C 180,E1 -24392.077,E2 -24392.077} C_VEL
LIN {X 0,Y 140.865,Z 537.999,A -85,B 0,C 180,E1 -24395.727,E2 -24395.727} C_VEL
LIN {X 0,Y 141.839,Z 536.326,A -85,B 0,C 180,E1 -24401.431,E2 -24401.431} C_VEL
LIN {X 0,Y 143.733,Z 533.5,A -85,B 0,C 180,E1 -24407.06,E2 -24407.06} C_VEL
LIN {X 0,Y 146.816,Z 529.444,A -85,B 0,C 180,E1 -24412.516,E2 -24412.516} C_VEL
LIN {X 0,Y 151.063,Z 523.901,A -85,B 0,C 180,E1 -24417.877,E2 -24417.877} C_VEL
LIN {X 0,Y 156.139,Z 517.198,A -85,B 0,C 180,E1 -24422.692,E2 -24422.692} C_VEL
LIN {X 0,Y 162.353,Z 508.624,A -85,B 0,C 180,E1 -24427.302,E2 -24427.302} C_VEL
LIN {X 0,Y 167.669,Z 500.91,A -85,B 0,C 180,E1 -24430.518,E2 -24430.518} C_VEL
LIN {X 0,Y 173.348,Z 491.827,A -85,B 0,C 180,E1 -24433.568,E2 -24433.568} C_VEL
LIN {X 0,Y 179.62,Z 481.101,A -85,B 0,C 180,E1 -24436.372,E2 -24436.372} C_VEL
LIN {X 0,Y 185.04,Z 470.56,A -85,B 0,C 180,E1 -24438.599,E2 -24438.599} C_VEL
LIN {X 0,Y 190.779,Z 458.014,A -85,B 0,C 180,E1 -24440.677,E2 -24440.677} C_VEL
LIN {X 0,Y 195.946,Z 444.405,A -85,B 0,C 180,E1 -24442.474,E2 -24442.474} C_VEL
LIN {X 0,Y 200.228,Z 430.937,A -85,B 0,C 180,E1 -24443.831,E2 -24443.831} C_VEL
LIN {X 0,Y 203.908,Z 416.287,A -85,B 0,C 180,E1 -24444.941,E2 -24444.941} C_VEL
LIN {X 0,Y 206.68,Z 401.577,A -85,B 0,C 180,E1 -24445.72,E2 -24445.72} C_VEL
LIN {X 0,Y 208.546,Z 385.983,A -85,B 0,C 180,E1 -24446.26,E2 -24446.26} C_VEL
LIN {X 0,Y 212.903,Z 332.491,A -85,B 0,C 180,E1 -24447.718,E2 -24447.718} C_VEL
LIN {X 0,Y 208.016,Z 322.789,A -85,B 0,C 180,E1 -24450.597,E2 -24450.597} C_VEL
LIN {X 0,Y 203.238,Z 314.213,A -85,B 0,C 180,E1 -24453.771,E2 -24453.771} C_VEL
LIN {X 0,Y 199.006,Z 307.357,A -85,B 0,C 180,E1 -24457.003,E2 -24457.003} C_VEL
LIN {X 0,Y 196.446,Z 303.456,A -85,B 0,C 180,E1 -24459.243,E2 -24459.243} C_VEL
LIN {X 0,Y 194.629,Z 300.61,A -85,B 0,C 180,E1 -24461.035,E2 -24461.035} C_VEL
LIN {X 0,Y 191.959,Z 296.663,A -85,B 0,C 180,E1 -24464.062,E2 -24464.062} C_VEL
LIN {X 0,Y 189.637,Z 293.221,A -85,B 0,C 180,E1 -24467.356,E2 -24467.356} C_VEL
LIN {X 0,Y 189.155,Z 292.272,A -85,B 0,C 180,E1 -24468.208,E2 -24468.208} C_VEL
LIN {X 0,Y 187.076,Z 289.817,A -85,B 0,C 180,E1 -24472.58,E2 -24472.58} C_VEL
LIN {X 0,Y 186.264,Z 287.28,A -85,B 0,C 180,E1 -24476.214,E2 -24476.214} C_VEL
LIN {X 0,Y 185.935,Z 286.954,A -85,B 0,C 180,E1 -24480,E2 -24480} C_VEL
LIN {X 0,Y 186.324,Z 287.406,A -85,B 0,C 180,E1 -24483.785,E2 -24483.785} C_VEL
LIN {X 0,Y 187.903,Z 291.137,A -85,B 0,C 180,E1 -24489.146,E2 -24489.146} C_VEL
LIN {X 0,Y 189.421,Z 292.757,A -85,B 0,C 180,E1 -24491.91,E2 -24491.91} C_VEL
LIN {X 0,Y 191.974,Z 296.627,A -85,B 0,C 180,E1 -24495.595,E2 -24495.595} C_VEL
LIN {X 0,Y 195.628,Z 302.1,A -85,B 0,C 180,E1 -24499.613,E2 -24499.613} C_VEL
LIN {X 0,Y 198.512,Z 306.606,A -85,B 0,C 180,E1 -24502.233,E2 -24502.233} C_VEL
LIN {X 0,Y 201.566,Z 311.492,A -85,B 0,C 180,E1 -24504.661,E2 -24504.661} C_VEL
LIN {X 0,Y 206.093,Z 321.161,A -85,B 0,C 180,E1 -24507.962,E2 -24507.962} C_VEL
LIN {X 0,Y 210.843,Z 332.647,A -85,B 0,C 180,E1 -24511.036,E2 -24511.036} C_VEL
LIN {X 0,Y 212.56,Z 337.257,A -85,B 0,C 180,E1 -24512.078,E2 -24512.078} C_VEL
LIN {X 0,Y 207.204,Z 400.864,A -85,B 0,C 180,E1 -24513.843,E2 -24513.843} C_VEL
LIN {X 0,Y 204.663,Z 416.468,A -85,B 0,C 180,E1 -24514.5,E2 -24514.5} C_VEL
LIN {X 0,Y 201.118,Z 431.695,A -85,B 0,C 180,E1 -24515.449,E2 -24515.449} C_VEL
LIN {X 0,Y 196.948,Z 445.418,A -85,B 0,C 180,E1 -24516.594,E2 -24516.594} C_VEL
LIN {X 0,Y 192.012,Z 458.867,A -85,B 0,C 180,E1 -24518.101,E2 -24518.101} C_VEL
LIN {X 0,Y 186.421,Z 471.884,A -85,B 0,C 180,E1 -24520.013,E2 -24520.013} C_VEL
LIN {X 0,Y 182.3,Z 480.328,A -85,B 0,C 180,E1 -24521.535,E2 -24521.535} C_VEL
LIN {X 0,Y 179.419,Z 484.92,A -85,B 0,C 180,E1 -24522.309,E2 -24522.309} C_VEL
LIN {X 0,Y 168.258,Z 497.591,A -85,B 0,C 180,E1 -24524.208,E2 -24524.208} C_VEL
LIN {X 0,Y 164.952,Z 501.563,A -85,B 0,C 180,E1 -24525.177,E2 -24525.177} C_VEL
LIN {X 0,Y 164.039,Z 502.847,A -85,B 0,C 180,E1 -24525.584,E2 -24525.584} C_VEL
LIN {X 0,Y 157.861,Z 511.798,A -85,B 0,C 180,E1 -24528.911,E2 -24528.911} C_VEL
LIN {X 0,Y 151.803,Z 520.195,A -85,B 0,C 180,E1 -24532.998,E2 -24532.998} C_VEL
LIN {X 0,Y 145.657,Z 528.018,A -85,B 0,C 180,E1 -24537.945,E2 -24537.945} C_VEL
LIN {X 0,Y 140.779,Z 534.253,A -85,B 0,C 180,E1 -24543.302,E2 -24543.302} C_VEL
LIN {X 0,Y 137.153,Z 539.084,A -85,B 0,C 180,E1 -24548.98,E2 -24548.98} C_VEL
LIN {X 0,Y 134.713,Z 542.63,A -85,B 0,C 180,E1 -24554.88,E2 -24554.88} C_VEL
LIN {X 0,Y 133.568,Z 544.974,A -85,B 0,C 180,E1 -24560.918,E2 -24560.918} C_VEL
LIN {X 0,Y 133.389,Z 546.159,A -85,B 0,C 180,E1 -24566.98,E2 -24566.98} C_VEL
LIN {X 0,Y 133.531,Z 546.318,A -85,B 0,C 180,E1 -24570,E2 -24570} C_VEL
LIN {X 0,Y 133.374,Z 545.691,A -85,B 0,C 180,E1 -24576.049,E2 -24576.049} C_VEL
LIN {X 0,Y 133.993,Z 543.906,A -85,B 0,C 180,E1 -24582.11,E2 -24582.11} C_VEL
LIN {X 0,Y 135.774,Z 540.949,A -85,B 0,C 180,E1 -24588.093,E2 -24588.093} C_VEL
LIN {X 0,Y 138.747,Z 536.753,A -85,B 0,C 180,E1 -24593.905,E2 -24593.905} C_VEL
LIN {X 0,Y 143.056,Z 531.211,A -85,B 0,C 180,E1 -24599.424,E2 -24599.424} C_VEL
LIN {X 0,Y 148.588,Z 524.175,A -85,B 0,C 180,E1 -24604.581,E2 -24604.581} C_VEL
LIN {X 0,Y 154.214,Z 516.654,A -85,B 0,C 180,E1 -24608.801,E2 -24608.801} C_VEL
LIN {X 0,Y 160.65,Z 507.595,A -85,B 0,C 180,E1 -24612.693,E2 -24612.693} C_VEL
LIN {X 0,Y 167.852,Z 496.715,A -85,B 0,C 180,E1 -24616.24,E2 -24616.24} C_VEL
LIN {X 0,Y 173.376,Z 487.476,A -85,B 0,C 180,E1 -24618.582,E2 -24618.582} C_VEL
LIN {X 0,Y 179.817,Z 475.606,A -85,B 0,C 180,E1 -24620.967,E2 -24620.967} C_VEL
LIN {X 0,Y 185.829,Z 462.618,A -85,B 0,C 180,E1 -24623.027,E2 -24623.027} C_VEL
LIN {X 0,Y 190.869,Z 450.037,A -85,B 0,C 180,E1 -24624.552,E2 -24624.552} C_VEL
LIN {X 0,Y 195.358,Z 436.504,A -85,B 0,C 180,E1 -24625.833,E2 -24625.833} C_VEL
LIN {X 0,Y 199.373,Z 421.516,A -85,B 0,C 180,E1 -24626.844,E2 -24626.844} C_VEL
LIN {X 0,Y 202.321,Z 406.268,A -85,B 0,C 180,E1 -24627.57,E2 -24627.57} C_VEL
LIN {X 0,Y 204.211,Z 390.067,A -85,B 0,C 180,E1 -24628.091,E2 -24628.091} C_VEL
LIN {X 0,Y 208.403,Z 339.807,A -85,B 0,C 180,E1 -24629.473,E2 -24629.473} C_VEL
LIN {X 0,Y 204.23,Z 329.005,A -85,B 0,C 180,E1 -24632.285,E2 -24632.285} C_VEL
LIN {X 0,Y 200.607,Z 320.425,A -85,B 0,C 180,E1 -24635.002,E2 -24635.002} C_VEL
LIN {X 0,Y 198.173,Z 315.599,A -85,B 0,C 180,E1 -24636.97,E2 -24636.97} C_VEL
LIN {X 0,Y 194.677,Z 309.942,A -85,B 0,C 180,E1 -24640.081,E2 -24640.081} C_VEL
LIN {X 0,Y 192.844,Z 307.059,A -85,B 0,C 180,E1 -24641.955,E2 -24641.955} C_VEL
LIN {X 0,Y 190.43,Z 303.304,A -85,B 0,C 180,E1 -24644.815,E2 -24644.815} C_VEL
LIN {X 0,Y 187.989,Z 299.321,A -85,B 0,C 180,E1 -24648.511,E2 -24648.511} C_VEL
LIN {X 0,Y 185.653,Z 296.108,A -85,B 0,C 180,E1 -24653.752,E2 -24653.752} C_VEL
LIN {X 0,Y 185.158,Z 294.242,A -85,B 0,C 180,E1 -24656.192,E2 -24656.192} C_VEL
LIN {X 0,Y 184.744,Z 293.892,A -85,B 0,C 180,E1 -24660,E2 -24660} C_VEL
LIN {X 0,Y 185.22,Z 294.456,A -85,B 0,C 180,E1 -24664.625,E2 -24664.625} C_VEL
LIN {X 0,Y 186.671,Z 297.997,A -85,B 0,C 180,E1 -24669.481,E2 -24669.481} C_VEL
LIN {X 0,Y 188.069,Z 299.518,A -85,B 0,C 180,E1 -24672.084,E2 -24672.084} C_VEL
LIN {X 0,Y 190.349,Z 303.211,A -85,B 0,C 180,E1 -24675.527,E2 -24675.527} C_VEL
LIN {X 0,Y 193.854,Z 308.573,A -85,B 0,C 180,E1 -24679.539,E2 -24679.539} C_VEL
LIN {X 0,Y 196.506,Z 312.914,A -85,B 0,C 180,E1 -24682.057,E2 -24682.057} C_VEL
LIN {X 0,Y 200.631,Z 319.879,A -85,B 0,C 180,E1 -24685.411,E2 -24685.411} C_VEL
LIN {X 0,Y 205.155,Z 328.288,A -85,B 0,C 180,E1 -24688.59,E2 -24688.59} C_VEL
LIN {X 0,Y 208.68,Z 335.45,A -85,B 0,C 180,E1 -24690.811,E2 -24690.811} C_VEL
LIN {X 0,Y 203.987,Z 390.817,A -85,B 0,C 180,E1 -24692.353,E2 -24692.353} C_VEL
LIN {X 0,Y 201.772,Z 406.284,A -85,B 0,C 180,E1 -24692.971,E2 -24692.971} C_VEL
LIN {X 0,Y 198.755,Z 420.498,A -85,B 0,C 180,E1 -24693.804,E2 -24693.804} C_VEL
LIN {X 0,Y 194.481,Z 435.695,A -85,B 0,C 180,E1 -24695.044,E2 -24695.044} C_VEL
LIN {X 0,Y 189.659,Z 449.668,A -85,B 0,C 180,E1 -24696.616,E2 -24696.616} C_VEL
LIN {X 0,Y 184.105,Z 462.868,A -85,B 0,C 180,E1 -24698.506,E2 -24698.506} C_VEL
LIN {X 0,Y 178.242,Z 474.652,A -85,B 0,C 180,E1 -24700.624,E2 -24700.624} C_VEL
LIN {X 0,Y 171.557,Z 486.455,A -85,B 0,C 180,E1 -24703.354,E2 -24703.354} C_VEL
LIN {X 0,Y 165.033,Z 496.681,A -85,B 0,C 180,E1 -24706.382,E2 -24706.382} C_VEL
LIN {X 0,Y 159.643,Z 504.805,A -85,B 0,C 180,E1 -24709.509,E2 -24709.509} C_VEL
LIN {X 0,Y 153.449,Z 513.056,A -85,B 0,C 180,E1 -24713.46,E2 -24713.46} C_VEL
LIN {X 0,Y 147.305,Z 520.8,A -85,B 0,C 180,E1 -24718.345,E2 -24718.345} C_VEL
LIN {X 0,Y 142.292,Z 526.955,A -85,B 0,C 180,E1 -24723.608,E2 -24723.608} C_VEL
LIN {X 0,Y 138.419,Z 531.7,A -85,B 0,C 180,E1 -24729.182,E2 -24729.182} C_VEL
LIN {X 0,Y 135.776,Z 535.166,A -85,B 0,C 180,E1 -24735.001,E2 -24735.001} C_VEL
LIN {X 0,Y 134.213,Z 537.45,A -85,B 0,C 180,E1 -24740.962,E2 -24740.962} C_VEL
LIN {X 0,Y 133.602,Z 538.607,A -85,B 0,C 180,E1 -24746.985,E2 -24746.985} C_VEL
LIN {X 0,Y 133.57,Z 538.703,A -85,B 0,C 180,E1 -24751.357,E2 -24751.357} C_VEL
LIN {X 0,Y 133.807,Z 538.199,A -85,B 0,C 180,E1 -24756.03,E2 -24756.03} C_VEL
LIN {X 0,Y 134.875,Z 536.527,A -85,B 0,C 180,E1 -24762.03,E2 -24762.03} C_VEL
LIN {X 0,Y 136.915,Z 533.701,A -85,B 0,C 180,E1 -24767.937,E2 -24767.937} C_VEL
LIN {X 0,Y 140.256,Z 529.644,A -85,B 0,C 180,E1 -24773.632,E2 -24773.632} C_VEL
LIN {X 0,Y 144.659,Z 524.263,A -85,B 0,C 180,E1 -24779.066,E2 -24779.066} C_VEL
LIN {X 0,Y 150.186,Z 517.398,A -85,B 0,C 180,E1 -24784.162,E2 -24784.162} C_VEL
LIN {X 0,Y 155.864,Z 510.017,A -85,B 0,C 180,E1 -24788.315,E2 -24788.315} C_VEL
LIN {X 0,Y 162.204,Z 501.257,A -85,B 0,C 180,E1 -24792.097,E2 -24792.097} C_VEL
LIN {X 0,Y 168.263,Z 492.026,A -85,B 0,C 180,E1 -24795.238,E2 -24795.238} C_VEL
LIN {X 0,Y 174.774,Z 481.3,A -85,B 0,C 180,E1 -24798.065,E2 -24798.065} C_VEL
LIN {X 0,Y 180.997,Z 469.588,A -85,B 0,C 180,E1 -24800.508,E2 -24800.508} C_VEL
LIN {X 0,Y 187.258,Z 456.082,A -85,B 0,C 180,E1 -24802.671,E2 -24802.671} C_VEL
LIN {X 0,Y 192.378,Z 442.66,A -85,B 0,C 180,E1 -24804.373,E2 -24804.373} C_VEL
LIN {X 0,Y 197.066,Z 427.748,A -85,B 0,C 180,E1 -24805.784,E2 -24805.784} C_VEL
LIN {X 0,Y 200.713,Z 412.675,A -85,B 0,C 180,E1 -24806.831,E2 -24806.831} C_VEL
LIN {X 0,Y 203.408,Z 397.431,A -85,B 0,C 180,E1 -24807.536,E2 -24807.536} C_VEL
LIN {X 0,Y 205.533,Z 376.291,A -85,B 0,C 180,E1 -24808.174,E2 -24808.174} C_VEL
LIN {X 0,Y 208.914,Z 335.694,A -85,B 0,C 180,E1 -24809.293,E2 -24809.293} C_VEL
LIN {X 0,Y 204.639,Z 327.057,A -85,B 0,C 180,E1 -24812.018,E2 -24812.018} C_VEL
LIN {X 0,Y 200.42,Z 319.246,A -85,B 0,C 180,E1 -24815.046,E2 -24815.046} C_VEL
LIN {X 0,Y 196.613,Z 312.926,A -85,B 0,C 180,E1 -24818.175,E2 -24818.175} C_VEL
LIN {X 0,Y 193.001,Z 307.134,A -85,B 0,C 180,E1 -24821.729,E2 -24821.729} C_VEL
LIN {X 0,Y 190.572,Z 303.372,A -85,B 0,C 180,E1 -24824.639,E2 -24824.639} C_VEL
LIN {X 0,Y 188.265,Z 299.68,A -85,B 0,C 180,E1 -24828.152,E2 -24828.152} C_VEL
LIN {X 0,Y 185.591,Z 295.402,A -85,B 0,C 180,E1 -24834.868,E2 -24834.868} C_VEL
LIN {X 0,Y 185.398,Z 294.349,A -85,B 0,C 180,E1 -24836.196,E2 -24836.196} C_VEL
LIN {X 0,Y 185.07,Z 294.002,A -85,B 0,C 180,E1 -24840,E2 -24840} C_VEL
LIN {X 0,Y 185.416,Z 294.573,A -85,B 0,C 180,E1 -24843.667,E2 -24843.667} C_VEL
LIN {X 0,Y 187.036,Z 298.284,A -85,B 0,C 180,E1 -24849.189,E2 -24849.189} C_VEL
LIN {X 0,Y 188.216,Z 299.593,A -85,B 0,C 180,E1 -24851.407,E2 -24851.407} C_VEL
LIN {X 0,Y 191.239,Z 304.379,A -85,B 0,C 180,E1 -24855.862,E2 -24855.862} C_VEL
LIN {X 0,Y 194.05,Z 308.764,A -85,B 0,C 180,E1 -24859.023,E2 -24859.023} C_VEL
LIN {X 0,Y 196.925,Z 313.452,A -85,B 0,C 180,E1 -24861.749,E2 -24861.749} C_VEL
LIN {X 0,Y 199.42,Z 317.698,A -85,B 0,C 180,E1 -24863.837,E2 -24863.837} C_VEL
LIN {X 0,Y 203.346,Z 326.475,A -85,B 0,C 180,E1 -24866.886,E2 -24866.886} C_VEL
LIN {X 0,Y 207.833,Z 337.833,A -85,B 0,C 180,E1 -24869.989,E2 -24869.989} C_VEL
LIN {X 0,Y 208.663,Z 340.077,A -85,B 0,C 180,E1 -24870.528,E2 -24870.528} C_VEL
LIN {X 0,Y 203.3,Z 400.964,A -85,B 0,C 180,E1 -24872.195,E2 -24872.195} C_VEL
LIN {X 0,Y 200.732,Z 416.277,A -85,B 0,C 180,E1 -24872.832,E2 -24872.832} C_VEL
LIN {X 0,Y 197.084,Z 431.501,A -85,B 0,C 180,E1 -24873.767,E2 -24873.767} C_VEL
LIN {X 0,Y 192.795,Z 445.223,A -85,B 0,C 180,E1 -24874.897,E2 -24874.897} C_VEL
LIN {X 0,Y 187.715,Z 458.671,A -85,B 0,C 180,E1 -24876.396,E2 -24876.396} C_VEL
LIN {X 0,Y 182.007,Z 471.522,A -85,B 0,C 180,E1 -24878.271,E2 -24878.271} C_VEL
LIN {X 0,Y 175.113,Z 484.781,A -85,B 0,C 180,E1 -24880.755,E2 -24880.755} C_VEL
LIN {X 0,Y 168.916,Z 495.188,A -85,B 0,C 180,E1 -24883.273,E2 -24883.273} C_VEL
LIN {X 0,Y 164.039,Z 502.847,A -85,B 0,C 180,E1 -24885.584,E2 -24885.584} C_VEL
LIN {X 0,Y 160.993,Z 506.683,A -85,B 0,C 180,E1 -24886.766,E2 -24886.766} C_VEL
LIN {X 0,Y 154.63,Z 512.613,A -85,B 0,C 180,E1 -24888.47,E2 -24888.47} C_VEL
LIN {X 0,Y 148.222,Z 518.128,A -85,B 0,C 180,E1 -24890.42,E2 -24890.42} C_VEL
LIN {X 0,Y 145.181,Z 521.19,A -85,B 0,C 180,E1 -24891.99,E2 -24891.99} C_VEL
LIN {X 0,Y 139.637,Z 527.816,A -85,B 0,C 180,E1 -24896.384,E2 -24896.384} C_VEL
LIN {X 0,Y 134.408,Z 534.051,A -85,B 0,C 180,E1 -24901.928,E2 -24901.928} C_VEL
LIN {X 0,Y 130.492,Z 538.882,A -85,B 0,C 180,E1 -24907.852,E2 -24907.852} C_VEL
LIN {X 0,Y 127.809,Z 542.428,A -85,B 0,C 180,E1 -24914.042,E2 -24914.042} C_VEL
LIN {X 0,Y 126.529,Z 544.772,A -85,B 0,C 180,E1 -24920.408,E2 -24920.408} C_VEL
LIN {X 0,Y 126.293,Z 545.958,A -85,B 0,C 180,E1 -24926.81,E2 -24926.81} C_VEL
LIN {X 0,Y 126.427,Z 546.117,A -85,B 0,C 180,E1 -24930,E2 -24930} C_VEL
LIN {X 0,Y 126.293,Z 545.952,A -85,B 0,C 180,E1 -24933.19,E2 -24933.19} C_VEL
LIN {X 0,Y 126.527,Z 544.741,A -85,B 0,C 180,E1 -24939.592,E2 -24939.592} C_VEL
LIN {X 0,Y 127.786,Z 542.373,A -85,B 0,C 180,E1 -24945.961,E2 -24945.961} C_VEL
LIN {X 0,Y 130.445,Z 538.808,A -85,B 0,C 180,E1 -24952.156,E2 -24952.156} C_VEL
LIN {X 0,Y 134.389,Z 533.955,A -85,B 0,C 180,E1 -24958.077,E2 -24958.077} C_VEL
LIN {X 0,Y 139.634,Z 527.686,A -85,B 0,C 180,E1 -24963.617,E2 -24963.617} C_VEL
LIN {X 0,Y 146.097,Z 519.828,A -85,B 0,C 180,E1 -24968.708,E2 -24968.708} C_VEL
LIN {X 0,Y 152.486,Z 511.476,A -85,B 0,C 180,E1 -24972.828,E2 -24972.828} C_VEL
LIN {X 0,Y 159.68,Z 501.421,A -85,B 0,C 180,E1 -24976.569,E2 -24976.569} C_VEL
LIN {X 0,Y 166.354,Z 491.152,A -85,B 0,C 180,E1 -24979.502,E2 -24979.502} C_VEL
LIN {X 0,Y 173.577,Z 478.914,A -85,B 0,C 180,E1 -24982.141,E2 -24982.141} C_VEL
LIN {X 0,Y 179.984,Z 466.063,A -85,B 0,C 180,E1 -24984.324,E2 -24984.324} C_VEL
LIN {X 0,Y 185.512,Z 453.25,A -85,B 0,C 180,E1 -24985.966,E2 -24985.966} C_VEL
LIN {X 0,Y 190.772,Z 438.477,A -85,B 0,C 180,E1 -24987.425,E2 -24987.425} C_VEL
LIN {X 0,Y 194.886,Z 424.162,A -85,B 0,C 180,E1 -24988.424,E2 -24988.424} C_VEL
LIN {X 0,Y 198.134,Z 408.925,A -85,B 0,C 180,E1 -24989.184,E2 -24989.184} C_VEL
LIN {X 0,Y 200.178,Z 393.732,A -85,B 0,C 180,E1 -24989.707,E2 -24989.707} C_VEL
LIN {X 0,Y 204.605,Z 342.59,A -85,B 0,C 180,E1 -24991.113,E2 -24991.113} C_VEL
LIN {X 0,Y 200.87,Z 332.71,A -85,B 0,C 180,E1 -24993.856,E2 -24993.856} C_VEL
LIN {X 0,Y 197.95,Z 325.52,A -85,B 0,C 180,E1 -24996.238,E2 -24996.238} C_VEL
LIN {X 0,Y 195.633,Z 320.86,A -85,B 0,C 180,E1 -24998.256,E2 -24998.256} C_VEL
LIN {X 0,Y 192.091,Z 314.894,A -85,B 0,C 180,E1 -25001.721,E2 -25001.721} C_VEL
LIN {X 0,Y 189.008,Z 309.932,A -85,B 0,C 180,E1 -25005.464,E2 -25005.464} C_VEL
LIN {X 0,Y 186.572,Z 305.924,A -85,B 0,C 180,E1 -25009.419,E2 -25009.419} C_VEL
LIN {X 0,Y 184.597,Z 302.826,A -85,B 0,C 180,E1 -25014.402,E2 -25014.402} C_VEL
LIN {X 0,Y 184.188,Z 301.215,A -85,B 0,C 180,E1 -25016.719,E2 -25016.719} C_VEL
LIN {X 0,Y 183.879,Z 300.941,A -85,B 0,C 180,E1 -25020,E2 -25020} C_VEL
LIN {X 0,Y 184.292,Z 301.505,A -85,B 0,C 180,E1 -25024.374,E2 -25024.374} C_VEL
LIN {X 0,Y 185.566,Z 304.848,A -85,B 0,C 180,E1 -25028.988,E2 -25028.988} C_VEL
LIN {X 0,Y 186.873,Z 306.367,A -85,B 0,C 180,E1 -25031.583,E2 -25031.583} C_VEL
LIN {X 0,Y 189.083,Z 310.043,A -85,B 0,C 180,E1 -25035.081,E2 -25035.081} C_VEL
LIN {X 0,Y 192.264,Z 315.21,A -85,B 0,C 180,E1 -25038.912,E2 -25038.912} C_VEL
LIN {X 0,Y 194.943,Z 319.805,A -85,B 0,C 180,E1 -25041.575,E2 -25041.575} C_VEL
LIN {X 0,Y 199.085,Z 327.113,A -85,B 0,C 180,E1 -25045.063,E2 -25045.063} C_VEL
LIN {X 0,Y 203.842,Z 336.596,A -85,B 0,C 180,E1 -25048.509,E2 -25048.509} C_VEL
LIN {X 0,Y 204.925,Z 338.913,A -85,B 0,C 180,E1 -25049.231,E2 -25049.231} C_VEL
LIN {X 0,Y 199.859,Z 394.77,A -85,B 0,C 180,E1 -25050.755,E2 -25050.755} C_VEL
LIN {X 0,Y 197.215,Z 410.658,A -85,B 0,C 180,E1 -25051.458,E2 -25051.458} C_VEL
LIN {X 0,Y 193.581,Z 425.738,A -85,B 0,C 180,E1 -25052.427,E2 -25052.427} C_VEL
LIN {X 0,Y 189.445,Z 439.159,A -85,B 0,C 180,E1 -25053.61,E2 -25053.61} C_VEL
LIN {X 0,Y 184.307,Z 452.984,A -85,B 0,C 180,E1 -25055.26,E2 -25055.26} C_VEL
LIN {X 0,Y 177.919,Z 466.886,A -85,B 0,C 180,E1 -25057.35,E2 -25057.35} C_VEL
LIN {X 0,Y 171.371,Z 479.083,A -85,B 0,C 180,E1 -25059.742,E2 -25059.742} C_VEL
LIN {X 0,Y 164.514,Z 490.198,A -85,B 0,C 180,E1 -25062.532,E2 -25062.532} C_VEL
LIN {X 0,Y 158.134,Z 499.577,A -85,B 0,C 180,E1 -25065.6,E2 -25065.6} C_VEL
LIN {X 0,Y 152.318,Z 507.493,A -85,B 0,C 180,E1 -25068.892,E2 -25068.892} C_VEL
LIN {X 0,Y 145.231,Z 516.343,A -85,B 0,C 180,E1 -25073.645,E2 -25073.645} C_VEL
LIN {X 0,Y 139.828,Z 522.669,A -85,B 0,C 180,E1 -25078.147,E2 -25078.147} C_VEL
LIN {X 0,Y 134.829,Z 528.469,A -85,B 0,C 180,E1 -25083.701,E2 -25083.701} C_VEL
LIN {X 0,Y 131.789,Z 531.902,A -85,B 0,C 180,E1 -25088.082,E2 -25088.082} C_VEL
LIN {X 0,Y 128.918,Z 535.368,A -85,B 0,C 180,E1 -25094.183,E2 -25094.183} C_VEL
LIN {X 0,Y 127.19,Z 537.651,A -85,B 0,C 180,E1 -25100.458,E2 -25100.458} C_VEL
LIN {X 0,Y 126.513,Z 538.808,A -85,B 0,C 180,E1 -25106.816,E2 -25106.816} C_VEL
LIN {X 0,Y 126.505,Z 538.961,A -85,B 0,C 180,E1 -25110,E2 -25110} C_VEL
LIN {X 0,Y 126.743,Z 538.4,A -85,B 0,C 180,E1 -25116.367,E2 -25116.367} C_VEL
LIN {X 0,Y 127.913,Z 536.728,A -85,B 0,C 180,E1 -25122.695,E2 -25122.695} C_VEL
LIN {X 0,Y 130.136,Z 533.902,A -85,B 0,C 180,E1 -25128.906,E2 -25128.906} C_VEL
LIN {X 0,Y 133.753,Z 529.845,A -85,B 0,C 180,E1 -25134.856,E2 -25134.856} C_VEL
LIN {X 0,Y 138.468,Z 524.463,A -85,B 0,C 180,E1 -25140.5,E2 -25140.5} C_VEL
LIN {X 0,Y 144.342,Z 517.598,A -85,B 0,C 180,E1 -25145.751,E2 -25145.751} C_VEL
LIN {X 0,Y 151.261,Z 509.023,A -85,B 0,C 180,E1 -25150.576,E2 -25150.576} C_VEL
LIN {X 0,Y 156.807,Z 501.689,A -85,B 0,C 180,E1 -25153.751,E2 -25153.751} C_VEL
LIN {X 0,Y 163.33,Z 492.224,A -85,B 0,C 180,E1 -25157.011,E2 -25157.011} C_VEL
LIN {X 0,Y 170.08,Z 481.499,A -85,B 0,C 180,E1 -25159.857,E2 -25159.857} C_VEL
LIN {X 0,Y 176.572,Z 469.785,A -85,B 0,C 180,E1 -25162.284,E2 -25162.284} C_VEL
LIN {X 0,Y 182.977,Z 456.418,A -85,B 0,C 180,E1 -25164.419,E2 -25164.419} C_VEL
LIN {X 0,Y 188.338,Z 442.855,A -85,B 0,C 180,E1 -25166.125,E2 -25166.125} C_VEL
LIN {X 0,Y 192.85,Z 429.069,A -85,B 0,C 180,E1 -25167.428,E2 -25167.428} C_VEL
LIN {X 0,Y 196.762,Z 413.626,A -85,B 0,C 180,E1 -25168.512,E2 -25168.512} C_VEL
LIN {X 0,Y 199.639,Z 397.957,A -85,B 0,C 180,E1 -25169.241,E2 -25169.241} C_VEL
LIN {X 0,Y 201.785,Z 377.664,A -85,B 0,C 180,E1 -25169.85,E2 -25169.85} C_VEL
LIN {X 0,Y 205.135,Z 339.08,A -85,B 0,C 180,E1 -25170.892,E2 -25170.892} C_VEL
LIN {X 0,Y 200.867,Z 330.286,A -85,B 0,C 180,E1 -25173.873,E2 -25173.873} C_VEL
LIN {X 0,Y 197.477,Z 323.959,A -85,B 0,C 180,E1 -25176.537,E2 -25176.537} C_VEL
LIN {X 0,Y 193.832,Z 317.587,A -85,B 0,C 180,E1 -25179.85,E2 -25179.85} C_VEL
LIN {X 0,Y 191.238,Z 313.386,A -85,B 0,C 180,E1 -25182.627,E2 -25182.627} C_VEL
LIN {X 0,Y 189.122,Z 309.976,A -85,B 0,C 180,E1 -25185.335,E2 -25185.335} C_VEL
LIN {X 0,Y 186.818,Z 306.045,A -85,B 0,C 180,E1 -25189.158,E2 -25189.158} C_VEL
LIN {X 0,Y 184.963,Z 303.356,A -85,B 0,C 180,E1 -25193.738,E2 -25193.738} C_VEL
LIN {X 0,Y 184.441,Z 301.316,A -85,B 0,C 180,E1 -25196.723,E2 -25196.723} C_VEL
LIN {X 0,Y 184.207,Z 301.026,A -85,B 0,C 180,E1 -25200,E2 -25200} C_VEL
LIN {X 0,Y 184.483,Z 301.499,A -85,B 0,C 180,E1 -25203.276,E2 -25203.276} C_VEL
LIN {X 0,Y 186.046,Z 305.287,A -85,B 0,C 180,E1 -25208.964,E2 -25208.964} C_VEL
LIN {X 0,Y 187.06,Z 306.493,A -85,B 0,C 180,E1 -25210.964,E2 -25210.964} C_VEL
LIN {X 0,Y 189.752,Z 310.922,A -85,B 0,C 180,E1 -25215.164,E2 -25215.164} C_VEL
LIN {X 0,Y 192.549,Z 315.502,A -85,B 0,C 180,E1 -25218.482,E2 -25218.482} C_VEL
LIN {X 0,Y 195.567,Z 320.605,A -85,B 0,C 180,E1 -25221.448,E2 -25221.448} C_VEL
LIN {X 0,Y 197.596,Z 324.51,A -85,B 0,C 180,E1 -25223.239,E2 -25223.239} C_VEL
LIN {X 0,Y 200.701,Z 331.86,A -85,B 0,C 180,E1 -25225.803,E2 -25225.803} C_VEL
LIN {X 0,Y 204.812,Z 342.794,A -85,B 0,C 180,E1 -25228.855,E2 -25228.855} C_VEL
LIN {X 0,Y 202.703,Z 367.581,A -85,B 0,C 180,E1 -25229.546,E2 -25229.546} C_VEL
LIN {X 0,Y 199.538,Z 401.205,A -85,B 0,C 180,E1 -25230.482,E2 -25230.482} C_VEL
LIN {X 0,Y 196.968,Z 416.086,A -85,B 0,C 180,E1 -25231.094,E2 -25231.094} C_VEL
LIN {X 0,Y 193.226,Z 431.307,A -85,B 0,C 180,E1 -25232.016,E2 -25232.016} C_VEL
LIN {X 0,Y 188.812,Z 445.028,A -85,B 0,C 180,E1 -25233.125,E2 -25233.125} C_VEL
LIN {X 0,Y 183.579,Z 458.475,A -85,B 0,C 180,E1 -25234.607,E2 -25234.607} C_VEL
LIN {X 0,Y 177.243,Z 472.232,A -85,B 0,C 180,E1 -25236.611,E2 -25236.611} C_VEL
LIN {X 0,Y 170.533,Z 484.582,A -85,B 0,C 180,E1 -25238.935,E2 -25238.935} C_VEL
LIN {X 0,Y 164.101,Z 494.989,A -85,B 0,C 180,E1 -25241.457,E2 -25241.457} C_VEL
LIN {X 0,Y 157.574,Z 504.657,A -85,B 0,C 180,E1 -25244.471,E2 -25244.471} C_VEL
LIN {X 0,Y 150.374,Z 514.377,A -85,B 0,C 180,E1 -25248.399,E2 -25248.399} C_VEL
LIN {X 0,Y 145.181,Z 521.19,A -85,B 0,C 180,E1 -25251.99,E2 -25251.99} C_VEL
LIN {X 0,Y 142.181,Z 524.154,A -85,B 0,C 180,E1 -25253.665,E2 -25253.665} C_VEL
LIN {X 0,Y 135.916,Z 528.602,A -85,B 0,C 180,E1 -25256.257,E2 -25256.257} C_VEL
LIN {X 0,Y 129.891,Z 532.536,A -85,B 0,C 180,E1 -25259.183,E2 -25259.183} C_VEL
LIN {X 0,Y 127.359,Z 534.671,A -85,B 0,C 180,E1 -25261.352,E2 -25261.352} C_VEL
LIN {X 0,Y 123.889,Z 538.68,A -85,B 0,C 180,E1 -25266.604,E2 -25266.604} C_VEL
LIN {X 0,Y 120.935,Z 542.226,A -85,B 0,C 180,E1 -25273.108,E2 -25273.108} C_VEL
LIN {X 0,Y 119.479,Z 544.57,A -85,B 0,C 180,E1 -25279.836,E2 -25279.836} C_VEL
LIN {X 0,Y 119.181,Z 545.757,A -85,B 0,C 180,E1 -25286.619,E2 -25286.619} C_VEL
LIN {X 0,Y 119.332,Z 545.917,A -85,B 0,C 180,E1 -25290,E2 -25290} C_VEL
LIN {X 0,Y 119.204,Z 545.287,A -85,B 0,C 180,E1 -25296.772,E2 -25296.772} C_VEL
LIN {X 0,Y 120.035,Z 543.5,A -85,B 0,C 180,E1 -25303.544,E2 -25303.544} C_VEL
LIN {X 0,Y 122.232,Z 540.543,A -85,B 0,C 180,E1 -25310.18,E2 -25310.18} C_VEL
LIN {X 0,Y 125.799,Z 536.281,A -85,B 0,C 180,E1 -25316.637,E2 -25316.637} C_VEL
LIN {X 0,Y 130.739,Z 530.802,A -85,B 0,C 180,E1 -25322.517,E2 -25322.517} C_VEL
LIN {X 0,Y 137.069,Z 523.768,A -85,B 0,C 180,E1 -25327.971,E2 -25327.971} C_VEL
LIN {X 0,Y 143.317,Z 516.259,A -85,B 0,C 180,E1 -25332.385,E2 -25332.385} C_VEL
LIN {X 0,Y 150.455,Z 507.186,A -85,B 0,C 180,E1 -25336.387,E2 -25336.387} C_VEL
LIN {X 0,Y 158.298,Z 496.305,A -85,B 0,C 180,E1 -25339.982,E2 -25339.982} C_VEL
LIN {X 0,Y 165.524,Z 485.109,A -85,B 0,C 180,E1 -25342.758,E2 -25342.758} C_VEL
LIN {X 0,Y 172.487,Z 472.798,A -85,B 0,C 180,E1 -25345.101,E2 -25345.101} C_VEL
LIN {X 0,Y 178.272,Z 460.775,A -85,B 0,C 180,E1 -25346.9,E2 -25346.9} C_VEL
LIN {X 0,Y 183.643,Z 447.854,A -85,B 0,C 180,E1 -25348.374,E2 -25348.374} C_VEL
LIN {X 0,Y 188.475,Z 433.831,A -85,B 0,C 180,E1 -25349.574,E2 -25349.574} C_VEL
LIN {X 0,Y 192.517,Z 418.807,A -85,B 0,C 180,E1 -25350.507,E2 -25350.507} C_VEL
LIN {X 0,Y 195.463,Z 403.226,A -85,B 0,C 180,E1 -25351.19,E2 -25351.19} C_VEL
LIN {X 0,Y 197.736,Z 382.361,A -85,B 0,C 180,E1 -25351.786,E2 -25351.786} C_VEL
LIN {X 0,Y 200.981,Z 346.276,A -85,B 0,C 180,E1 -25352.745,E2 -25352.745} C_VEL
LIN {X 0,Y 200.797,Z 345.113,A -85,B 0,C 180,E1 -25352.935,E2 -25352.935} C_VEL
LIN {X 0,Y 197.464,Z 335.854,A -85,B 0,C 180,E1 -25355.656,E2 -25355.656} C_VEL
LIN {X 0,Y 194.668,Z 328.965,A -85,B 0,C 180,E1 -25358.177,E2 -25358.177} C_VEL
LIN {X 0,Y 191.517,Z 323.261,A -85,B 0,C 180,E1 -25361.271,E2 -25361.271} C_VEL
LIN {X 0,Y 189.5,Z 319.84,A -85,B 0,C 180,E1 -25363.574,E2 -25363.574} C_VEL
LIN {X 0,Y 187.515,Z 316.453,A -85,B 0,C 180,E1 -25366.257,E2 -25366.257} C_VEL
LIN {X 0,Y 185.421,Z 312.783,A -85,B 0,C 180,E1 -25369.904,E2 -25369.904} C_VEL
LIN {X 0,Y 183.607,Z 309.704,A -85,B 0,C 180,E1 -25374.853,E2 -25374.853} C_VEL
LIN {X 0,Y 183.319,Z 308.301,A -85,B 0,C 180,E1 -25376.704,E2 -25376.704} C_VEL
LIN {X 0,Y 183.014,Z 307.986,A -85,B 0,C 180,E1 -25380,E2 -25380} C_VEL
LIN {X 0,Y 183.35,Z 308.457,A -85,B 0,C 180,E1 -25383.984,E2 -25383.984} C_VEL
LIN {X 0,Y 184.698,Z 311.998,A -85,B 0,C 180,E1 -25389.031,E2 -25389.031} C_VEL
LIN {X 0,Y 185.733,Z 313.286,A -85,B 0,C 180,E1 -25391.156,E2 -25391.156} C_VEL
LIN {X 0,Y 188.19,Z 317.58,A -85,B 0,C 180,E1 -25395.154,E2 -25395.154} C_VEL
LIN {X 0,Y 190.682,Z 321.833,A -85,B 0,C 180,E1 -25398.258,E2 -25398.258} C_VEL
LIN {X 0,Y 193.869,Z 327.422,A -85,B 0,C 180,E1 -25401.522,E2 -25401.522} C_VEL
LIN {X 0,Y 197.477,Z 334.351,A -85,B 0,C 180,E1 -25404.667,E2 -25404.667} C_VEL
LIN {X 0,Y 201.241,Z 342.222,A -85,B 0,C 180,E1 -25407.533,E2 -25407.533} C_VEL
LIN {X 0,Y 196.418,Z 394.357,A -85,B 0,C 180,E1 -25408.956,E2 -25408.956} C_VEL
LIN {X 0,Y 193.791,Z 410.1,A -85,B 0,C 180,E1 -25409.631,E2 -25409.631} C_VEL
LIN {X 0,Y 189.876,Z 425.945,A -85,B 0,C 180,E1 -25410.622,E2 -25410.622} C_VEL
LIN {X 0,Y 185.224,Z 440.441,A -85,B 0,C 180,E1 -25411.901,E2 -25411.901} C_VEL
LIN {X 0,Y 180.158,Z 453.499,A -85,B 0,C 180,E1 -25413.452,E2 -25413.452} C_VEL
LIN {X 0,Y 173.709,Z 467.091,A -85,B 0,C 180,E1 -25415.491,E2 -25415.491} C_VEL
LIN {X 0,Y 166.897,Z 479.288,A -85,B 0,C 180,E1 -25417.857,E2 -25417.857} C_VEL
LIN {X 0,Y 159.785,Z 490.402,A -85,B 0,C 180,E1 -25420.649,E2 -25420.649} C_VEL
LIN {X 0,Y 152.633,Z 500.473,A -85,B 0,C 180,E1 -25423.988,E2 -25423.988} C_VEL
LIN {X 0,Y 147.036,Z 507.697,A -85,B 0,C 180,E1 -25427.07,E2 -25427.07} C_VEL
LIN {X 0,Y 139.536,Z 516.547,A -85,B 0,C 180,E1 -25431.904,E2 -25431.904} C_VEL
LIN {X 0,Y 133.822,Z 522.872,A -85,B 0,C 180,E1 -25436.535,E2 -25436.535} C_VEL
LIN {X 0,Y 128.446,Z 528.673,A -85,B 0,C 180,E1 -25442.285,E2 -25442.285} C_VEL
LIN {X 0,Y 125.216,Z 532.105,A -85,B 0,C 180,E1 -25446.866,E2 -25446.866} C_VEL
LIN {X 0,Y 122.077,Z 535.57,A -85,B 0,C 180,E1 -25453.271,E2 -25453.271} C_VEL
LIN {X 0,Y 120.193,Z 537.853,A -85,B 0,C 180,E1 -25459.897,E2 -25459.897} C_VEL
LIN {X 0,Y 119.437,Z 539.009,A -85,B 0,C 180,E1 -25466.627,E2 -25466.627} C_VEL
LIN {X 0,Y 119.419,Z 539.161,A -85,B 0,C 180,E1 -25470,E2 -25470} C_VEL
LIN {X 0,Y 119.683,Z 538.601,A -85,B 0,C 180,E1 -25476.744,E2 -25476.744} C_VEL
LIN {X 0,Y 120.982,Z 536.929,A -85,B 0,C 180,E1 -25483.436,E2 -25483.436} C_VEL
LIN {X 0,Y 123.402,Z 534.104,A -85,B 0,C 180,E1 -25489.981,E2 -25489.981} C_VEL
LIN {X 0,Y 127.32,Z 530.046,A -85,B 0,C 180,E1 -25496.205,E2 -25496.205} C_VEL
LIN {X 0,Y 132.367,Z 524.664,A -85,B 0,C 180,E1 -25502.069,E2 -25502.069} C_VEL
LIN {X 0,Y 138.617,Z 517.799,A -85,B 0,C 180,E1 -25507.474,E2 -25507.474} C_VEL
LIN {X 0,Y 145.934,Z 509.222,A -85,B 0,C 180,E1 -25512.393,E2 -25512.393} C_VEL
LIN {X 0,Y 151.559,Z 502.108,A -85,B 0,C 180,E1 -25515.527,E2 -25515.527} C_VEL
LIN {X 0,Y 158.564,Z 492.423,A -85,B 0,C 180,E1 -25518.892,E2 -25518.892} C_VEL
LIN {X 0,Y 165.573,Z 481.697,A -85,B 0,C 180,E1 -25521.743,E2 -25521.743} C_VEL
LIN {X 0,Y 172.317,Z 469.983,A -85,B 0,C 180,E1 -25524.154,E2 -25524.154} C_VEL
LIN {X 0,Y 178.873,Z 456.755,A -85,B 0,C 180,E1 -25526.25,E2 -25526.25} C_VEL
LIN {X 0,Y 184.476,Z 443.05,A -85,B 0,C 180,E1 -25527.956,E2 -25527.956} C_VEL
LIN {X 0,Y 189.44,Z 428.136,A -85,B 0,C 180,E1 -25529.34,E2 -25529.34} C_VEL
LIN {X 0,Y 193.332,Z 413.055,A -85,B 0,C 180,E1 -25530.345,E2 -25530.345} C_VEL
